// TwinCAT 3 PLC project PlanarTrackMovement_1
// ProgramVersion: 3.1.4026.12
// libraries:
//   HelperFunctions, * (Amazon)
//   RingBuffer, * (Amazon)
//   Tc2_Standard, * (Beckhoff Automation GmbH)
//   Tc2_System, * (Beckhoff Automation GmbH)
//   Tc2_Utilities, * (Beckhoff Automation GmbH)
//   Tc3_Mc3PlanarMotion, * (Beckhoff Automation GmbH)
//   Tc3_Module, * (Beckhoff Automation GmbH)
//   Tc3_Physics, * (Beckhoff Automation GmbH)
//   Tc3_XTS_Utility, * (Beckhoff Automation GmbH)
// project tree:
//   DUTs/ E_MergeType.TcDUT, E_TrackNum.TcDUT, MoverSort.TcDUT, ST_Debounce.TcDUT, ST_MoverOptions.TcDUT, ST_PlanarTrackConfig.TcDUT, ST_DivertConfig.TcDUT, ST_ExpMoverStatus.TcDUT, ST_PlcSystem.TcDUT, ST_SectorsConfig.TcDUT, ST_SectorsStatus.TcDUT, ST_SwitchStatus.TcDUT, ST_SectorConfig.TcDUT, ST_SectorStatus.TcDUT, ST_ShortcutConfig.TcDUT, ST_SwitchConfig.TcDUT, ST_TrackConfig.TcDUT, ST_MoverConfig.TcDUT
//   GVLs/ GC.TcGVL, GVL_General.TcGVL, GVL_Mc3.TcGVL
//   ITFs/ I_Mover.TcIO, I_MoverSector.TcIO
//   / PlcTask.TcTTO
//   POUs/FBs/ FB_AllTrackSectors.TcPOU, FB_AllExpMovers.TcPOU, FB_DivertQueue.TcPOU, FB_ExpandedMover.TcPOU, FB_MoverLists.TcPOU, FB_MoveState.TcPOU, FB_RobMover.TcPOU (excluded from build), FB_PlanarXtsMover.TcPOU, FB_PWM.TcPOU (not stored), FB_TrackSector.TcPOU, FB_SwitchMagnet.TcPOU, FB_TrackSectors.TcPOU, ReadTcCom.TcPOU
//   POUs/FUNs/ F_CurrentVelocity.TcPOU, F_PosnInitial.TcPOU, F_PosnDisp.TcPOU, F_t_SL2a.TcPOU, F_t_v0.TcPOU, F_t_vConstant.TcPOU, IsBetween.TcPOU (not stored), PositionF_CurrentCoeff.TcPOU
//   POUs/ MAIN.TcPOU
// real-time tasks:
//   TASK XTS Task: cycle T#500us, priority 1, ADS port 350
//   TASK Job Task: cycle default, priority 32
//   TASK MC-Task (MET): cycle T#2ms, priority 3, ADS port 521
//   TASK MC-Task (MPT): cycle T#10ms, priority 8, ADS port 531
//   TASK PlcTask: cycle T#1ms, priority 20, ADS port 351
//   TASK PlcTask1: cycle T#1ms, priority 21, ADS port 352
// motion (NC):
//   TASK NC-Task 1 SAF: cycle T#2ms, priority 4, ADS port 501
//   TASK NC-Task 1 SVB: cycle T#10ms, priority 9, ADS port 511
//   AXIS Axis 1 (id 1)
//     General: UnitFlags=#x00000004
//     Dynamic: Acceleration=4000, Deceleration=4000, Jerk=10000
//     Velo: FastManual=1200, Maximum=5000
//     OtherSettings: AllowMotionCmdToSlave=true
//     encoder EncType=28
//       EncPara: MaxCount=#xffffffff
//     drive DrvType=22
//       DrvPara: MaxCount=#xffffffff, DriveControlDWord=#x00000100
//         Analog: VeloReferenz=5000, TorqueSetpointScale=10, ScaleFactorActTorque=0.1
//         TimeComp: TaskDelayCycles=1
//     controller CtrType=1
//       CtrPara: PriorControlFactor=1
//         PosDiffControl: Range=50
//         Observer: BandWidth=20
// I/O:
//   DEVICE Device 1 (EtherCAT) (disabled), AmsNetId 11.200.5.30.2.1
//     Term 1 (EK1200) [EK1200-5000 EtherCAT Power supply (2A E-Bus)]
//       Term 2 (EL1809) [EL1809 16Ch. Dig. Input 24V, 3ms]
//       Term 3 (EL1018) [EL1018 8Ch. Dig. Input 24V, 10µs]
//       Term 4 (EL2809) [EL2809 16Ch. Dig. Output 24V, 0.5A]
//       Term 5 (EL3004) [EL3004 4Ch. Ana. Input +/-10V]
//       Term 6 (EL3314) [EL3314 4Ch. Ana. Input Thermocouple (TC)]
//       Term 7 (EL4034) [EL4034 4Ch. Ana. Output +/-10V, 12bit]
//       Term 8 (EL7062) [EL7062-0000 Stepper Drive]
//       Term 9 (EL9576) [EL9576 Brake chopper terminal]
//       Term 10 (EL9410) [EL9410 E-Bus Power Supplier  (Diagnostics)]
//       Term 11 (EL1904) [EL1904, 4 Ch. Safety Input 24V, TwinSAFE]
//         modules: Module 1 (FSOES)
//       Term 12 (EL1904) [EL1904, 4 Ch. Safety Input 24V, TwinSAFE]
//         modules: Module 1 (FSOES)
//       Term 13 (EL2912) [EL2912, 2Ch. Safety Output 24V, 2A, TwinSAFE]
//         modules: Module 2 (FSOUT), Module 3 (DEVICEIO), Module 4 (FSLOGIC)
//       Term 14 (EK1122) [EK1122 2 port EtherCAT junction]
//       Term 95 (EL6695) [EL6695 EtherCAT Bridge terminal (Primary)]
//       Term 16 (EK1110) [EK1110 EtherCAT extension]
//     Term 15 (AX8640-0000-0105) [AX8640-0000-0105]
//       startup 32768:16 := 12 // PSM Parameters / Ext brake resistor overload factor at 1% duty cycle
//       startup 32768:18 := 21DCC63E // PSM Parameters / External brake resistor time constant 1
//       startup 32768:19 := C37C6442 // PSM Parameters / External brake resistor time constant 2
//       startup 32768:20 := 8CA3E13F // PSM Parameters / External brake resistor partial fraction factor
//   DEVICE Device 8 (EtherCAT) (disabled), AmsNetId 11.200.5.30.9.1
//     Box 18 (AT5100-0100) [AT5100-0100 XTS XL, TwinSAFE]
//       modules: Module 1 (SAFETY)
//     Box 19 (AT5100-0100) [AT5100-0100 XTS XL, TwinSAFE]
//       modules: Module 1 (SAFETY)
//     Box 20 (AT5100-0100) [AT5100-0100 XTS XL, TwinSAFE]
//       modules: Module 1 (SAFETY)
//     Box 21 (AT5100-0100) [AT5100-0100 XTS XL, TwinSAFE]
//       modules: Module 1 (SAFETY)
//     Box 22 (AT5100-0100) [AT5100-0100 XTS XL, TwinSAFE]
//       modules: Module 1 (SAFETY)
//     Box 23 (AT5100-0100) [AT5100-0100 XTS XL, TwinSAFE]
//       modules: Module 1 (SAFETY)
//     Box 24 (AT5100-0100) [AT5100-0100 XTS XL, TwinSAFE]
//       modules: Module 1 (SAFETY)
//     Box 25 (AT5100-0100) [AT5100-0100 XTS XL, TwinSAFE]
//       modules: Module 1 (SAFETY)
//     Box 26 (AT5100-0100) [AT5100-0100 XTS XL, TwinSAFE]
//       modules: Module 1 (SAFETY)
//     Box 27 (AT5100-0100) [AT5100-0100 XTS XL, TwinSAFE]
//       modules: Module 1 (SAFETY)
//     Box 28 (AT5100-0100) [AT5100-0100 XTS XL, TwinSAFE]
//       modules: Module 1 (SAFETY)
//     Box 29 (AT5100-0100) [AT5100-0100 XTS XL, TwinSAFE]
//       modules: Module 1 (SAFETY)
//     Box 30 (AT5100-0100) [AT5100-0100 XTS XL, TwinSAFE]
//       modules: Module 1 (SAFETY)
//     Box 31 (AT5100-0100) [AT5100-0100 XTS XL, TwinSAFE]
//       modules: Module 1 (SAFETY)
//     Box 32 (AT5100-0100) [AT5100-0100 XTS XL, TwinSAFE]
//       modules: Module 1 (SAFETY)
//     Box 33 (AT5100-0100) [AT5100-0100 XTS XL, TwinSAFE]
//       modules: Module 1 (SAFETY)
//     Box 34 (AT5100-0100) [AT5100-0100 XTS XL, TwinSAFE]
//       modules: Module 1 (SAFETY)
//     Box 35 (AT5100-0100) [AT5100-0100 XTS XL, TwinSAFE]
//       modules: Module 1 (SAFETY)
//     Box 36 (AT5100-0100) [AT5100-0100 XTS XL, TwinSAFE]
//       modules: Module 1 (SAFETY)
//     Box 37 (AT5100-0100) [AT5100-0100 XTS XL, TwinSAFE]
//       modules: Module 1 (SAFETY)
//     Box 38 (AT5100-0100) [AT5100-0100 XTS XL, TwinSAFE]
//       modules: Module 1 (SAFETY)
//     Box 39 (AT5100-0100) [AT5100-0100 XTS XL, TwinSAFE]
//       modules: Module 1 (SAFETY)
//     Box 40 (AT5100-0100) [AT5100-0100 XTS XL, TwinSAFE]
//       modules: Module 1 (SAFETY)
//     Box 41 (AT5100-0100) [AT5100-0100 XTS XL, TwinSAFE]
//       modules: Module 1 (SAFETY)
//     Box 42 (AT5100-0100) [AT5100-0100 XTS XL, TwinSAFE]
//       modules: Module 1 (SAFETY)
//     Box 43 (AT5100-0100) [AT5100-0100 XTS XL, TwinSAFE]
//       modules: Module 1 (SAFETY)
//     Box 44 (AT5100-0100) [AT5100-0100 XTS XL, TwinSAFE]
//       modules: Module 1 (SAFETY)
//     Box 45 (AT5100-0100) [AT5100-0100 XTS XL, TwinSAFE]
//       modules: Module 1 (SAFETY)
//     Box 46 (AT5100-0100) [AT5100-0100 XTS XL, TwinSAFE]
//       modules: Module 1 (SAFETY)
//     Box 47 (AT5100-0100) [AT5100-0100 XTS XL, TwinSAFE]
//       modules: Module 1 (SAFETY)
//     Box 48 (AT5100-0100) [AT5100-0100 XTS XL, TwinSAFE]
//       modules: Module 1 (SAFETY)
//     Box 49 (AT5100-0100) [AT5100-0100 XTS XL, TwinSAFE]
//       modules: Module 1 (SAFETY)
//   DEVICE Device 4 (EtherCAT) (disabled), AmsNetId 11.200.5.30.5.1
//     Box 50 (AT5100-0100) [AT5100-0100 XTS XL, TwinSAFE]
//       modules: Module 1 (SAFETY)
//     Box 51 (AT5100-0100) [AT5100-0100 XTS XL, TwinSAFE]
//       modules: Module 1 (SAFETY)
//     Box 52 (AT5100-0100) [AT5100-0100 XTS XL, TwinSAFE]
//       modules: Module 1 (SAFETY)
//     Box 53 (AT5100-0100) [AT5100-0100 XTS XL, TwinSAFE]
//       modules: Module 1 (SAFETY)
//     Box 54 (AT5100-0100) [AT5100-0100 XTS XL, TwinSAFE]
//       modules: Module 1 (SAFETY)
//     Box 55 (AT5100-0100) [AT5100-0100 XTS XL, TwinSAFE]
//       modules: Module 1 (SAFETY)
//     Box 56 (AT5100-0100) [AT5100-0100 XTS XL, TwinSAFE]
//       modules: Module 1 (SAFETY)
//     Box 57 (AT5100-0100) [AT5100-0100 XTS XL, TwinSAFE]
//       modules: Module 1 (SAFETY)
//     Box 58 (AT5100-0100) [AT5100-0100 XTS XL, TwinSAFE]
//       modules: Module 1 (SAFETY)
//     Box 59 (AT5100-0100) [AT5100-0100 XTS XL, TwinSAFE]
//       modules: Module 1 (SAFETY)
//     Box 60 (AT5100-0100) [AT5100-0100 XTS XL, TwinSAFE]
//       modules: Module 1 (SAFETY)
//     Box 61 (AT5100-0100) [AT5100-0100 XTS XL, TwinSAFE]
//       modules: Module 1 (SAFETY)
//     Box 62 (AT5100-0100) [AT5100-0100 XTS XL, TwinSAFE]
//       modules: Module 1 (SAFETY)
//     Box 63 (AT5100-0100) [AT5100-0100 XTS XL, TwinSAFE]
//       modules: Module 1 (SAFETY)
//     Box 64 (AT5100-0100) [AT5100-0100 XTS XL, TwinSAFE]
//       modules: Module 1 (SAFETY)
//     Box 65 (AT5100-0100) [AT5100-0100 XTS XL, TwinSAFE]
//       modules: Module 1 (SAFETY)
//     Box 66 (AT5100-0100) [AT5100-0100 XTS XL, TwinSAFE]
//       modules: Module 1 (SAFETY)
//     Box 67 (AT5100-0100) [AT5100-0100 XTS XL, TwinSAFE]
//       modules: Module 1 (SAFETY)
//     Box 68 (AT5100-0100) [AT5100-0100 XTS XL, TwinSAFE]
//       modules: Module 1 (SAFETY)
//     Box 69 (AT5100-0100) [AT5100-0100 XTS XL, TwinSAFE]
//       modules: Module 1 (SAFETY)
//     Box 70 (AT5100-0100) [AT5100-0100 XTS XL, TwinSAFE]
//       modules: Module 1 (SAFETY)
//     Box 71 (AT5100-0100) [AT5100-0100 XTS XL, TwinSAFE]
//       modules: Module 1 (SAFETY)
//     Box 72 (AT5100-0100) [AT5100-0100 XTS XL, TwinSAFE]
//       modules: Module 1 (SAFETY)
//     Box 73 (AT5100-0100) [AT5100-0100 XTS XL, TwinSAFE]
//       modules: Module 1 (SAFETY)
//     Box 74 (AT5100-0100) [AT5100-0100 XTS XL, TwinSAFE]
//       modules: Module 1 (SAFETY)
//     Box 75 (AT5100-0100) [AT5100-0100 XTS XL, TwinSAFE]
//       modules: Module 1 (SAFETY)
//     Box 76 (AT5100-0100) [AT5100-0100 XTS XL, TwinSAFE]
//       modules: Module 1 (SAFETY)
//     Box 77 (AT5100-0100) [AT5100-0100 XTS XL, TwinSAFE]
//       modules: Module 1 (SAFETY)
//     Box 78 (AT5100-0100) [AT5100-0100 XTS XL, TwinSAFE]
//       modules: Module 1 (SAFETY)
//     Box 79 (AT5100-0100) [AT5100-0100 XTS XL, TwinSAFE]
//       modules: Module 1 (SAFETY)
//     Box 80 (AT5100-0100) [AT5100-0100 XTS XL, TwinSAFE]
//       modules: Module 1 (SAFETY)
//     Box 81 (AT5100-0100) [AT5100-0100 XTS XL, TwinSAFE]
//       modules: Module 1 (SAFETY)
// variable links:
//   Device 1 (EtherCAT) <-> Device 1 (EtherCAT)/Term 1 (EK1200)/Term 12 (EL1904)
//     Term 1 (EK1200)/Term 13 (EL2912)/ConnectionInputs/TwinSafeGroup1.Term 12 (EL1904) - Module 1 (FSOES)_144 TxPDO <-> Module 1 (FSOES)/RxPDO/FSOE
//   Device 1 (EtherCAT) <-> Device 1 (EtherCAT)/Term 1 (EK1200)/Term 13 (EL2912)
//     Term 1 (EK1200)/Term 11 (EL1904)/Module 1 (FSOES)/RxPDO/FSOE <-> ConnectionInputs/TwinSafeGroup1.Term 11 (EL1904) - Module 1 (FSOES)_4 TxPDO
//     Term 1 (EK1200)/Term 11 (EL1904)/Module 1 (FSOES)/TxPDO/FSOE <-> ConnectionOutputs/TwinSafeGroup1.Term 11 (EL1904) - Module 1 (FSOES)_4 RxPDO
//     Term 1 (EK1200)/Term 12 (EL1904)/Module 1 (FSOES)/TxPDO/FSOE <-> ConnectionOutputs/TwinSafeGroup1.Term 12 (EL1904) - Module 1 (FSOES)_144 RxPDO
//   Device 1 (EtherCAT) <-> Device 4 (EtherCAT)/Box 50 (AT5100-0100)
//     Term 1 (EK1200)/Term 13 (EL2912)/ConnectionInputs/TwinSafeGroup1.Box 50 (AT5100-0100) - Module 1 (SAFETY)_107 TxPDO <-> Module 1 (SAFETY)/SAFETY FSoE Connection 1 Receive Message/Message_4
//     Term 1 (EK1200)/Term 13 (EL2912)/ConnectionOutputs/TwinSafeGroup1.Box 50 (AT5100-0100) - Module 1 (SAFETY)_107 RxPDO <-> Module 1 (SAFETY)/SAFETY FSoE Connection 1 Send Message/Message_4
//   Device 1 (EtherCAT) <-> Device 4 (EtherCAT)/Box 51 (AT5100-0100)
//     Term 1 (EK1200)/Term 13 (EL2912)/ConnectionInputs/TwinSafeGroup1.Box 51 (AT5100-0100) - Module 1 (SAFETY)_108 TxPDO <-> Module 1 (SAFETY)/SAFETY FSoE Connection 1 Receive Message/Message_4
//     Term 1 (EK1200)/Term 13 (EL2912)/ConnectionOutputs/TwinSafeGroup1.Box 51 (AT5100-0100) - Module 1 (SAFETY)_108 RxPDO <-> Module 1 (SAFETY)/SAFETY FSoE Connection 1 Send Message/Message_4
//   Device 1 (EtherCAT) <-> Device 4 (EtherCAT)/Box 52 (AT5100-0100)
//     Term 1 (EK1200)/Term 13 (EL2912)/ConnectionInputs/TwinSafeGroup1.Box 52 (AT5100-0100) - Module 1 (SAFETY)_109 TxPDO <-> Module 1 (SAFETY)/SAFETY FSoE Connection 1 Receive Message/Message_4
//     Term 1 (EK1200)/Term 13 (EL2912)/ConnectionOutputs/TwinSafeGroup1.Box 52 (AT5100-0100) - Module 1 (SAFETY)_109 RxPDO <-> Module 1 (SAFETY)/SAFETY FSoE Connection 1 Send Message/Message_4
//   Device 1 (EtherCAT) <-> Device 4 (EtherCAT)/Box 53 (AT5100-0100)
//     Term 1 (EK1200)/Term 13 (EL2912)/ConnectionInputs/TwinSafeGroup1.Box 53 (AT5100-0100) - Module 1 (SAFETY)_110 TxPDO <-> Module 1 (SAFETY)/SAFETY FSoE Connection 1 Receive Message/Message_4
//     Term 1 (EK1200)/Term 13 (EL2912)/ConnectionOutputs/TwinSafeGroup1.Box 53 (AT5100-0100) - Module 1 (SAFETY)_110 RxPDO <-> Module 1 (SAFETY)/SAFETY FSoE Connection 1 Send Message/Message_4
//   Device 1 (EtherCAT) <-> Device 4 (EtherCAT)/Box 54 (AT5100-0100)
//     Term 1 (EK1200)/Term 13 (EL2912)/ConnectionInputs/TwinSafeGroup1.Box 54 (AT5100-0100) - Module 1 (SAFETY)_111 TxPDO <-> Module 1 (SAFETY)/SAFETY FSoE Connection 1 Receive Message/Message_4
//     Term 1 (EK1200)/Term 13 (EL2912)/ConnectionOutputs/TwinSafeGroup1.Box 54 (AT5100-0100) - Module 1 (SAFETY)_111 RxPDO <-> Module 1 (SAFETY)/SAFETY FSoE Connection 1 Send Message/Message_4
//   Device 1 (EtherCAT) <-> Device 4 (EtherCAT)/Box 55 (AT5100-0100)
//     Term 1 (EK1200)/Term 13 (EL2912)/ConnectionInputs/TwinSafeGroup1.Box 55 (AT5100-0100) - Module 1 (SAFETY)_112 TxPDO <-> Module 1 (SAFETY)/SAFETY FSoE Connection 1 Receive Message/Message_4
//     Term 1 (EK1200)/Term 13 (EL2912)/ConnectionOutputs/TwinSafeGroup1.Box 55 (AT5100-0100) - Module 1 (SAFETY)_112 RxPDO <-> Module 1 (SAFETY)/SAFETY FSoE Connection 1 Send Message/Message_4
//   Device 1 (EtherCAT) <-> Device 4 (EtherCAT)/Box 56 (AT5100-0100)
//     Term 1 (EK1200)/Term 13 (EL2912)/ConnectionInputs/TwinSafeGroup1.Box 56 (AT5100-0100) - Module 1 (SAFETY)_113 TxPDO <-> Module 1 (SAFETY)/SAFETY FSoE Connection 1 Receive Message/Message_4
//     Term 1 (EK1200)/Term 13 (EL2912)/ConnectionOutputs/TwinSafeGroup1.Box 56 (AT5100-0100) - Module 1 (SAFETY)_113 RxPDO <-> Module 1 (SAFETY)/SAFETY FSoE Connection 1 Send Message/Message_4
//   Device 1 (EtherCAT) <-> Device 4 (EtherCAT)/Box 57 (AT5100-0100)
//     Term 1 (EK1200)/Term 13 (EL2912)/ConnectionInputs/TwinSafeGroup1.Box 57 (AT5100-0100) - Module 1 (SAFETY)_114 TxPDO <-> Module 1 (SAFETY)/SAFETY FSoE Connection 1 Receive Message/Message_4
//     Term 1 (EK1200)/Term 13 (EL2912)/ConnectionOutputs/TwinSafeGroup1.Box 57 (AT5100-0100) - Module 1 (SAFETY)_114 RxPDO <-> Module 1 (SAFETY)/SAFETY FSoE Connection 1 Send Message/Message_4
//   Device 1 (EtherCAT) <-> Device 4 (EtherCAT)/Box 58 (AT5100-0100)
//     Term 1 (EK1200)/Term 13 (EL2912)/ConnectionInputs/TwinSafeGroup1.Box 58 (AT5100-0100) - Module 1 (SAFETY)_115 TxPDO <-> Module 1 (SAFETY)/SAFETY FSoE Connection 1 Receive Message/Message_4
//     Term 1 (EK1200)/Term 13 (EL2912)/ConnectionOutputs/TwinSafeGroup1.Box 58 (AT5100-0100) - Module 1 (SAFETY)_115 RxPDO <-> Module 1 (SAFETY)/SAFETY FSoE Connection 1 Send Message/Message_4
//   Device 1 (EtherCAT) <-> Device 4 (EtherCAT)/Box 59 (AT5100-0100)
//     Term 1 (EK1200)/Term 13 (EL2912)/ConnectionOutputs/TwinSafeGroup1.Box 59 (AT5100-0100) - Module 1 (SAFETY)_116 RxPDO <-> Module 1 (SAFETY)/SAFETY FSoE Connection 1 Send Message/Message_4
//   Device 1 (EtherCAT) <-> Device 4 (EtherCAT)/Box 60 (AT5100-0100)
//     Term 1 (EK1200)/Term 13 (EL2912)/ConnectionInputs/TwinSafeGroup1.Box 60 (AT5100-0100) - Module 1 (SAFETY)_117 TxPDO <-> Module 1 (SAFETY)/SAFETY FSoE Connection 1 Receive Message/Message_4
//     Term 1 (EK1200)/Term 13 (EL2912)/ConnectionOutputs/TwinSafeGroup1.Box 60 (AT5100-0100) - Module 1 (SAFETY)_117 RxPDO <-> Module 1 (SAFETY)/SAFETY FSoE Connection 1 Send Message/Message_4
//   Device 1 (EtherCAT) <-> Device 4 (EtherCAT)/Box 61 (AT5100-0100)
//     Term 1 (EK1200)/Term 13 (EL2912)/ConnectionInputs/TwinSafeGroup1.Box 61 (AT5100-0100) - Module 1 (SAFETY)_118 TxPDO <-> Module 1 (SAFETY)/SAFETY FSoE Connection 1 Receive Message/Message_4
//   Device 1 (EtherCAT) <-> Device 4 (EtherCAT)/Box 62 (AT5100-0100)
//     Term 1 (EK1200)/Term 13 (EL2912)/ConnectionInputs/TwinSafeGroup1.Box 62 (AT5100-0100) - Module 1 (SAFETY)_119 TxPDO <-> Module 1 (SAFETY)/SAFETY FSoE Connection 1 Receive Message/Message_4
//   Device 1 (EtherCAT) <-> Device 4 (EtherCAT)/Box 63 (AT5100-0100)
//     Term 1 (EK1200)/Term 13 (EL2912)/ConnectionInputs/TwinSafeGroup1.Box 63 (AT5100-0100) - Module 1 (SAFETY)_120 TxPDO <-> Module 1 (SAFETY)/SAFETY FSoE Connection 1 Receive Message/Message_4
//     Term 1 (EK1200)/Term 13 (EL2912)/ConnectionOutputs/TwinSafeGroup1.Box 63 (AT5100-0100) - Module 1 (SAFETY)_120 RxPDO <-> Module 1 (SAFETY)/SAFETY FSoE Connection 1 Send Message/Message_4
//   Device 1 (EtherCAT) <-> Device 4 (EtherCAT)/Box 64 (AT5100-0100)
//     Term 1 (EK1200)/Term 13 (EL2912)/ConnectionInputs/TwinSafeGroup1.Box 64 (AT5100-0100) - Module 1 (SAFETY)_121 TxPDO <-> Module 1 (SAFETY)/SAFETY FSoE Connection 1 Receive Message/Message_4
//     Term 1 (EK1200)/Term 13 (EL2912)/ConnectionOutputs/TwinSafeGroup1.Box 64 (AT5100-0100) - Module 1 (SAFETY)_121 RxPDO <-> Module 1 (SAFETY)/SAFETY FSoE Connection 1 Send Message/Message_4
//   Device 1 (EtherCAT) <-> Device 4 (EtherCAT)/Box 65 (AT5100-0100)
//     Term 1 (EK1200)/Term 13 (EL2912)/ConnectionInputs/TwinSafeGroup1.Box 65 (AT5100-0100) - Module 1 (SAFETY)_122 TxPDO <-> Module 1 (SAFETY)/SAFETY FSoE Connection 1 Receive Message/Message_4
//     Term 1 (EK1200)/Term 13 (EL2912)/ConnectionOutputs/TwinSafeGroup1.Box 65 (AT5100-0100) - Module 1 (SAFETY)_122 RxPDO <-> Module 1 (SAFETY)/SAFETY FSoE Connection 1 Send Message/Message_4
//   Device 1 (EtherCAT) <-> Device 4 (EtherCAT)/Box 66 (AT5100-0100)
//     Term 1 (EK1200)/Term 13 (EL2912)/ConnectionInputs/TwinSafeGroup1.Box 66 (AT5100-0100) - Module 1 (SAFETY)_123 TxPDO <-> Module 1 (SAFETY)/SAFETY FSoE Connection 1 Receive Message/Message_4
//     Term 1 (EK1200)/Term 13 (EL2912)/ConnectionOutputs/TwinSafeGroup1.Box 66 (AT5100-0100) - Module 1 (SAFETY)_123 RxPDO <-> Module 1 (SAFETY)/SAFETY FSoE Connection 1 Send Message/Message_4
//   Device 1 (EtherCAT) <-> Device 4 (EtherCAT)/Box 67 (AT5100-0100)
//     Term 1 (EK1200)/Term 13 (EL2912)/ConnectionInputs/TwinSafeGroup1.Box 67 (AT5100-0100) - Module 1 (SAFETY)_124 TxPDO <-> Module 1 (SAFETY)/SAFETY FSoE Connection 1 Receive Message/Message_4
//     Term 1 (EK1200)/Term 13 (EL2912)/ConnectionOutputs/TwinSafeGroup1.Box 67 (AT5100-0100) - Module 1 (SAFETY)_124 RxPDO <-> Module 1 (SAFETY)/SAFETY FSoE Connection 1 Send Message/Message_4
//   Device 1 (EtherCAT) <-> Device 4 (EtherCAT)/Box 68 (AT5100-0100)
//     Term 1 (EK1200)/Term 13 (EL2912)/ConnectionInputs/TwinSafeGroup1.Box 68 (AT5100-0100) - Module 1 (SAFETY)_125 TxPDO <-> Module 1 (SAFETY)/SAFETY FSoE Connection 1 Receive Message/Message_4
//     Term 1 (EK1200)/Term 13 (EL2912)/ConnectionOutputs/TwinSafeGroup1.Box 68 (AT5100-0100) - Module 1 (SAFETY)_125 RxPDO <-> Module 1 (SAFETY)/SAFETY FSoE Connection 1 Send Message/Message_4
//   Device 1 (EtherCAT) <-> Device 4 (EtherCAT)/Box 69 (AT5100-0100)
//     Term 1 (EK1200)/Term 13 (EL2912)/ConnectionInputs/TwinSafeGroup1.Box 69 (AT5100-0100) - Module 1 (SAFETY)_126 TxPDO <-> Module 1 (SAFETY)/SAFETY FSoE Connection 1 Receive Message/Message_4
//     Term 1 (EK1200)/Term 13 (EL2912)/ConnectionOutputs/TwinSafeGroup1.Box 69 (AT5100-0100) - Module 1 (SAFETY)_126 RxPDO <-> Module 1 (SAFETY)/SAFETY FSoE Connection 1 Send Message/Message_4
//   Device 1 (EtherCAT) <-> Device 4 (EtherCAT)/Box 70 (AT5100-0100)
//     Term 1 (EK1200)/Term 13 (EL2912)/ConnectionInputs/TwinSafeGroup1.Box 70 (AT5100-0100) - Module 1 (SAFETY)_127 TxPDO <-> Module 1 (SAFETY)/SAFETY FSoE Connection 1 Receive Message/Message_4
//     Term 1 (EK1200)/Term 13 (EL2912)/ConnectionOutputs/TwinSafeGroup1.Box 70 (AT5100-0100) - Module 1 (SAFETY)_127 RxPDO <-> Module 1 (SAFETY)/SAFETY FSoE Connection 1 Send Message/Message_4
//   Device 1 (EtherCAT) <-> Device 4 (EtherCAT)/Box 71 (AT5100-0100)
//     Term 1 (EK1200)/Term 13 (EL2912)/ConnectionInputs/TwinSafeGroup1.Box 71 (AT5100-0100) - Module 1 (SAFETY)_128 TxPDO <-> Module 1 (SAFETY)/SAFETY FSoE Connection 1 Receive Message/Message_4
//     Term 1 (EK1200)/Term 13 (EL2912)/ConnectionOutputs/TwinSafeGroup1.Box 71 (AT5100-0100) - Module 1 (SAFETY)_128 RxPDO <-> Module 1 (SAFETY)/SAFETY FSoE Connection 1 Send Message/Message_4
//   Device 1 (EtherCAT) <-> Device 4 (EtherCAT)/Box 72 (AT5100-0100)
//     Term 1 (EK1200)/Term 13 (EL2912)/ConnectionInputs/TwinSafeGroup1.Box 72 (AT5100-0100) - Module 1 (SAFETY)_129 TxPDO <-> Module 1 (SAFETY)/SAFETY FSoE Connection 1 Receive Message/Message_4
//     Term 1 (EK1200)/Term 13 (EL2912)/ConnectionOutputs/TwinSafeGroup1.Box 72 (AT5100-0100) - Module 1 (SAFETY)_129 RxPDO <-> Module 1 (SAFETY)/SAFETY FSoE Connection 1 Send Message/Message_4
//   Device 1 (EtherCAT) <-> Device 4 (EtherCAT)/Box 73 (AT5100-0100)
//     Term 1 (EK1200)/Term 13 (EL2912)/ConnectionInputs/TwinSafeGroup1.Box 73 (AT5100-0100) - Module 1 (SAFETY)_130 TxPDO <-> Module 1 (SAFETY)/SAFETY FSoE Connection 1 Receive Message/Message_4
//     Term 1 (EK1200)/Term 13 (EL2912)/ConnectionOutputs/TwinSafeGroup1.Box 73 (AT5100-0100) - Module 1 (SAFETY)_130 RxPDO <-> Module 1 (SAFETY)/SAFETY FSoE Connection 1 Send Message/Message_4
//   Device 1 (EtherCAT) <-> Device 4 (EtherCAT)/Box 74 (AT5100-0100)
//     Term 1 (EK1200)/Term 13 (EL2912)/ConnectionOutputs/TwinSafeGroup1.Box 74 (AT5100-0100) - Module 1 (SAFETY)_131 RxPDO <-> Module 1 (SAFETY)/SAFETY FSoE Connection 1 Send Message/Message_4
//   Device 1 (EtherCAT) <-> Device 4 (EtherCAT)/Box 75 (AT5100-0100)
//     Term 1 (EK1200)/Term 13 (EL2912)/ConnectionInputs/TwinSafeGroup1.Box 75 (AT5100-0100) - Module 1 (SAFETY)_132 TxPDO <-> Module 1 (SAFETY)/SAFETY FSoE Connection 1 Receive Message/Message_4
//     Term 1 (EK1200)/Term 13 (EL2912)/ConnectionOutputs/TwinSafeGroup1.Box 75 (AT5100-0100) - Module 1 (SAFETY)_132 RxPDO <-> Module 1 (SAFETY)/SAFETY FSoE Connection 1 Send Message/Message_4
//   Device 1 (EtherCAT) <-> Device 4 (EtherCAT)/Box 76 (AT5100-0100)
//     Term 1 (EK1200)/Term 13 (EL2912)/ConnectionInputs/TwinSafeGroup1.Box 76 (AT5100-0100) - Module 1 (SAFETY)_133 TxPDO <-> Module 1 (SAFETY)/SAFETY FSoE Connection 1 Receive Message/Message_4
//     Term 1 (EK1200)/Term 13 (EL2912)/ConnectionOutputs/TwinSafeGroup1.Box 76 (AT5100-0100) - Module 1 (SAFETY)_133 RxPDO <-> Module 1 (SAFETY)/SAFETY FSoE Connection 1 Send Message/Message_4
//   Device 1 (EtherCAT) <-> Device 4 (EtherCAT)/Box 77 (AT5100-0100)
//     Term 1 (EK1200)/Term 13 (EL2912)/ConnectionInputs/TwinSafeGroup1.Box 77 (AT5100-0100) - Module 1 (SAFETY)_134 TxPDO <-> Module 1 (SAFETY)/SAFETY FSoE Connection 1 Receive Message/Message_4
//     Term 1 (EK1200)/Term 13 (EL2912)/ConnectionOutputs/TwinSafeGroup1.Box 77 (AT5100-0100) - Module 1 (SAFETY)_134 RxPDO <-> Module 1 (SAFETY)/SAFETY FSoE Connection 1 Send Message/Message_4
//   Device 1 (EtherCAT) <-> Device 4 (EtherCAT)/Box 78 (AT5100-0100)
//     Term 1 (EK1200)/Term 13 (EL2912)/ConnectionInputs/TwinSafeGroup1.Box 78 (AT5100-0100) - Module 1 (SAFETY)_135 TxPDO <-> Module 1 (SAFETY)/SAFETY FSoE Connection 1 Receive Message/Message_4
//     Term 1 (EK1200)/Term 13 (EL2912)/ConnectionOutputs/TwinSafeGroup1.Box 78 (AT5100-0100) - Module 1 (SAFETY)_135 RxPDO <-> Module 1 (SAFETY)/SAFETY FSoE Connection 1 Send Message/Message_4
//   Device 1 (EtherCAT) <-> Device 4 (EtherCAT)/Box 79 (AT5100-0100)
//     Term 1 (EK1200)/Term 13 (EL2912)/ConnectionInputs/TwinSafeGroup1.Box 79 (AT5100-0100) - Module 1 (SAFETY)_136 TxPDO <-> Module 1 (SAFETY)/SAFETY FSoE Connection 1 Receive Message/Message_4
//     Term 1 (EK1200)/Term 13 (EL2912)/ConnectionOutputs/TwinSafeGroup1.Box 79 (AT5100-0100) - Module 1 (SAFETY)_136 RxPDO <-> Module 1 (SAFETY)/SAFETY FSoE Connection 1 Send Message/Message_4
//   Device 1 (EtherCAT) <-> Device 4 (EtherCAT)/Box 80 (AT5100-0100)
//     Term 1 (EK1200)/Term 13 (EL2912)/ConnectionInputs/TwinSafeGroup1.Box 80 (AT5100-0100) - Module 1 (SAFETY)_137 TxPDO <-> Module 1 (SAFETY)/SAFETY FSoE Connection 1 Receive Message/Message_4
//     Term 1 (EK1200)/Term 13 (EL2912)/ConnectionOutputs/TwinSafeGroup1.Box 80 (AT5100-0100) - Module 1 (SAFETY)_137 RxPDO <-> Module 1 (SAFETY)/SAFETY FSoE Connection 1 Send Message/Message_4
//   Device 1 (EtherCAT) <-> Device 4 (EtherCAT)/Box 81 (AT5100-0100)
//     Term 1 (EK1200)/Term 13 (EL2912)/ConnectionInputs/TwinSafeGroup1.Box 81 (AT5100-0100) - Module 1 (SAFETY)_138 TxPDO <-> Module 1 (SAFETY)/SAFETY FSoE Connection 1 Receive Message/Message_4
//     Term 1 (EK1200)/Term 13 (EL2912)/ConnectionOutputs/TwinSafeGroup1.Box 81 (AT5100-0100) - Module 1 (SAFETY)_138 RxPDO <-> Module 1 (SAFETY)/SAFETY FSoE Connection 1 Send Message/Message_4
//   Device 1 (EtherCAT) <-> Device 8 (EtherCAT)/Box 18 (AT5100-0100)
//     Term 1 (EK1200)/Term 13 (EL2912)/ConnectionInputs/TwinSafeGroup1.Box 18 (AT5100-0100) - Module 1 (SAFETY)_71 TxPDO <-> Module 1 (SAFETY)/SAFETY FSoE Connection 1 Receive Message/Message_4
//     Term 1 (EK1200)/Term 13 (EL2912)/ConnectionOutputs/TwinSafeGroup1.Box 18 (AT5100-0100) - Module 1 (SAFETY)_71 RxPDO <-> Module 1 (SAFETY)/SAFETY FSoE Connection 1 Send Message/Message_4
//   Device 1 (EtherCAT) <-> Device 8 (EtherCAT)/Box 19 (AT5100-0100)
//     Term 1 (EK1200)/Term 13 (EL2912)/ConnectionInputs/TwinSafeGroup1.Box 19 (AT5100-0100) - Module 1 (SAFETY)_76 TxPDO <-> Module 1 (SAFETY)/SAFETY FSoE Connection 1 Receive Message/Message_4
//     Term 1 (EK1200)/Term 13 (EL2912)/ConnectionOutputs/TwinSafeGroup1.Box 19 (AT5100-0100) - Module 1 (SAFETY)_76 RxPDO <-> Module 1 (SAFETY)/SAFETY FSoE Connection 1 Send Message/Message_4
//   Device 1 (EtherCAT) <-> Device 8 (EtherCAT)/Box 20 (AT5100-0100)
//     Term 1 (EK1200)/Term 13 (EL2912)/ConnectionInputs/TwinSafeGroup1.Box 20 (AT5100-0100) - Module 1 (SAFETY)_77 TxPDO <-> Module 1 (SAFETY)/SAFETY FSoE Connection 1 Receive Message/Message_4
//     Term 1 (EK1200)/Term 13 (EL2912)/ConnectionOutputs/TwinSafeGroup1.Box 20 (AT5100-0100) - Module 1 (SAFETY)_77 RxPDO <-> Module 1 (SAFETY)/SAFETY FSoE Connection 1 Send Message/Message_4
//   Device 1 (EtherCAT) <-> Device 8 (EtherCAT)/Box 21 (AT5100-0100)
//     Term 1 (EK1200)/Term 13 (EL2912)/ConnectionInputs/TwinSafeGroup1.Box 21 (AT5100-0100) - Module 1 (SAFETY)_78 TxPDO <-> Module 1 (SAFETY)/SAFETY FSoE Connection 1 Receive Message/Message_4
//     Term 1 (EK1200)/Term 13 (EL2912)/ConnectionOutputs/TwinSafeGroup1.Box 21 (AT5100-0100) - Module 1 (SAFETY)_78 RxPDO <-> Module 1 (SAFETY)/SAFETY FSoE Connection 1 Send Message/Message_4
//   Device 1 (EtherCAT) <-> Device 8 (EtherCAT)/Box 22 (AT5100-0100)
//     Term 1 (EK1200)/Term 13 (EL2912)/ConnectionInputs/TwinSafeGroup1.Box 22 (AT5100-0100) - Module 1 (SAFETY)_79 TxPDO <-> Module 1 (SAFETY)/SAFETY FSoE Connection 1 Receive Message/Message_4
//     Term 1 (EK1200)/Term 13 (EL2912)/ConnectionOutputs/TwinSafeGroup1.Box 22 (AT5100-0100) - Module 1 (SAFETY)_79 RxPDO <-> Module 1 (SAFETY)/SAFETY FSoE Connection 1 Send Message/Message_4
//   Device 1 (EtherCAT) <-> Device 8 (EtherCAT)/Box 23 (AT5100-0100)
//     Term 1 (EK1200)/Term 13 (EL2912)/ConnectionInputs/TwinSafeGroup1.Box 23 (AT5100-0100) - Module 1 (SAFETY)_80 TxPDO <-> Module 1 (SAFETY)/SAFETY FSoE Connection 1 Receive Message/Message_4
//     Term 1 (EK1200)/Term 13 (EL2912)/ConnectionOutputs/TwinSafeGroup1.Box 23 (AT5100-0100) - Module 1 (SAFETY)_80 RxPDO <-> Module 1 (SAFETY)/SAFETY FSoE Connection 1 Send Message/Message_4
//   Device 1 (EtherCAT) <-> Device 8 (EtherCAT)/Box 24 (AT5100-0100)
//     Term 1 (EK1200)/Term 13 (EL2912)/ConnectionOutputs/TwinSafeGroup1.Box 24 (AT5100-0100) - Module 1 (SAFETY)_81 RxPDO <-> Module 1 (SAFETY)/SAFETY FSoE Connection 1 Send Message/Message_4
//   Device 1 (EtherCAT) <-> Device 8 (EtherCAT)/Box 25 (AT5100-0100)
//     Term 1 (EK1200)/Term 13 (EL2912)/ConnectionInputs/TwinSafeGroup1.Box 25 (AT5100-0100) - Module 1 (SAFETY)_82 TxPDO <-> Module 1 (SAFETY)/SAFETY FSoE Connection 1 Receive Message/Message_4
//     Term 1 (EK1200)/Term 13 (EL2912)/ConnectionOutputs/TwinSafeGroup1.Box 25 (AT5100-0100) - Module 1 (SAFETY)_82 RxPDO <-> Module 1 (SAFETY)/SAFETY FSoE Connection 1 Send Message/Message_4
//   Device 1 (EtherCAT) <-> Device 8 (EtherCAT)/Box 26 (AT5100-0100)
//     Term 1 (EK1200)/Term 13 (EL2912)/ConnectionInputs/TwinSafeGroup1.Box 26 (AT5100-0100) - Module 1 (SAFETY)_83 TxPDO <-> Module 1 (SAFETY)/SAFETY FSoE Connection 1 Receive Message/Message_4
//     Term 1 (EK1200)/Term 13 (EL2912)/ConnectionOutputs/TwinSafeGroup1.Box 26 (AT5100-0100) - Module 1 (SAFETY)_83 RxPDO <-> Module 1 (SAFETY)/SAFETY FSoE Connection 1 Send Message/Message_4
//   Device 1 (EtherCAT) <-> Device 8 (EtherCAT)/Box 27 (AT5100-0100)
//     Term 1 (EK1200)/Term 13 (EL2912)/ConnectionInputs/TwinSafeGroup1.Box 27 (AT5100-0100) - Module 1 (SAFETY)_84 TxPDO <-> Module 1 (SAFETY)/SAFETY FSoE Connection 1 Receive Message/Message_4
//     Term 1 (EK1200)/Term 13 (EL2912)/ConnectionOutputs/TwinSafeGroup1.Box 27 (AT5100-0100) - Module 1 (SAFETY)_84 RxPDO <-> Module 1 (SAFETY)/SAFETY FSoE Connection 1 Send Message/Message_4
//   Device 1 (EtherCAT) <-> Device 8 (EtherCAT)/Box 28 (AT5100-0100)
//     Term 1 (EK1200)/Term 13 (EL2912)/ConnectionInputs/TwinSafeGroup1.Box 28 (AT5100-0100) - Module 1 (SAFETY)_85 TxPDO <-> Module 1 (SAFETY)/SAFETY FSoE Connection 1 Receive Message/Message_4
//     Term 1 (EK1200)/Term 13 (EL2912)/ConnectionOutputs/TwinSafeGroup1.Box 28 (AT5100-0100) - Module 1 (SAFETY)_85 RxPDO <-> Module 1 (SAFETY)/SAFETY FSoE Connection 1 Send Message/Message_4
//   Device 1 (EtherCAT) <-> Device 8 (EtherCAT)/Box 29 (AT5100-0100)
//     Term 1 (EK1200)/Term 13 (EL2912)/ConnectionInputs/TwinSafeGroup1.Box 29 (AT5100-0100) - Module 1 (SAFETY)_86 TxPDO <-> Module 1 (SAFETY)/SAFETY FSoE Connection 1 Receive Message/Message_4
//     Term 1 (EK1200)/Term 13 (EL2912)/ConnectionOutputs/TwinSafeGroup1.Box 29 (AT5100-0100) - Module 1 (SAFETY)_86 RxPDO <-> Module 1 (SAFETY)/SAFETY FSoE Connection 1 Send Message/Message_4
//   Device 1 (EtherCAT) <-> Device 8 (EtherCAT)/Box 30 (AT5100-0100)
//     Term 1 (EK1200)/Term 13 (EL2912)/ConnectionInputs/TwinSafeGroup1.Box 30 (AT5100-0100) - Module 1 (SAFETY)_87 TxPDO <-> Module 1 (SAFETY)/SAFETY FSoE Connection 1 Receive Message/Message_4
//     Term 1 (EK1200)/Term 13 (EL2912)/ConnectionOutputs/TwinSafeGroup1.Box 30 (AT5100-0100) - Module 1 (SAFETY)_87 RxPDO <-> Module 1 (SAFETY)/SAFETY FSoE Connection 1 Send Message/Message_4
//   Device 1 (EtherCAT) <-> Device 8 (EtherCAT)/Box 31 (AT5100-0100)
//     Term 1 (EK1200)/Term 13 (EL2912)/ConnectionInputs/TwinSafeGroup1.Box 31 (AT5100-0100) - Module 1 (SAFETY)_88 TxPDO <-> Module 1 (SAFETY)/SAFETY FSoE Connection 1 Receive Message/Message_4
//     Term 1 (EK1200)/Term 13 (EL2912)/ConnectionOutputs/TwinSafeGroup1.Box 31 (AT5100-0100) - Module 1 (SAFETY)_88 RxPDO <-> Module 1 (SAFETY)/SAFETY FSoE Connection 1 Send Message/Message_4
//   Device 1 (EtherCAT) <-> Device 8 (EtherCAT)/Box 32 (AT5100-0100)
//     Term 1 (EK1200)/Term 13 (EL2912)/ConnectionInputs/TwinSafeGroup1.Box 32 (AT5100-0100) - Module 1 (SAFETY)_89 TxPDO <-> Module 1 (SAFETY)/SAFETY FSoE Connection 1 Receive Message/Message_4
//     Term 1 (EK1200)/Term 13 (EL2912)/ConnectionOutputs/TwinSafeGroup1.Box 32 (AT5100-0100) - Module 1 (SAFETY)_89 RxPDO <-> Module 1 (SAFETY)/SAFETY FSoE Connection 1 Send Message/Message_4
//   Device 1 (EtherCAT) <-> Device 8 (EtherCAT)/Box 33 (AT5100-0100)
//     Term 1 (EK1200)/Term 13 (EL2912)/ConnectionInputs/TwinSafeGroup1.Box 33 (AT5100-0100) - Module 1 (SAFETY)_90 TxPDO <-> Module 1 (SAFETY)/SAFETY FSoE Connection 1 Receive Message/Message_4
//     Term 1 (EK1200)/Term 13 (EL2912)/ConnectionOutputs/TwinSafeGroup1.Box 33 (AT5100-0100) - Module 1 (SAFETY)_90 RxPDO <-> Module 1 (SAFETY)/SAFETY FSoE Connection 1 Send Message/Message_4
//   Device 1 (EtherCAT) <-> Device 8 (EtherCAT)/Box 34 (AT5100-0100)
//     Term 1 (EK1200)/Term 13 (EL2912)/ConnectionInputs/TwinSafeGroup1.Box 34 (AT5100-0100) - Module 1 (SAFETY)_91 TxPDO <-> Module 1 (SAFETY)/SAFETY FSoE Connection 1 Receive Message/Message_4
//     Term 1 (EK1200)/Term 13 (EL2912)/ConnectionOutputs/TwinSafeGroup1.Box 34 (AT5100-0100) - Module 1 (SAFETY)_91 RxPDO <-> Module 1 (SAFETY)/SAFETY FSoE Connection 1 Send Message/Message_4
//   Device 1 (EtherCAT) <-> Device 8 (EtherCAT)/Box 35 (AT5100-0100)
//     Term 1 (EK1200)/Term 13 (EL2912)/ConnectionInputs/TwinSafeGroup1.Box 35 (AT5100-0100) - Module 1 (SAFETY)_92 TxPDO <-> Module 1 (SAFETY)/SAFETY FSoE Connection 1 Receive Message/Message_4
//     Term 1 (EK1200)/Term 13 (EL2912)/ConnectionOutputs/TwinSafeGroup1.Box 35 (AT5100-0100) - Module 1 (SAFETY)_92 RxPDO <-> Module 1 (SAFETY)/SAFETY FSoE Connection 1 Send Message/Message_4
//   Device 1 (EtherCAT) <-> Device 8 (EtherCAT)/Box 36 (AT5100-0100)
//     Term 1 (EK1200)/Term 13 (EL2912)/ConnectionInputs/TwinSafeGroup1.Box 36 (AT5100-0100) - Module 1 (SAFETY)_93 TxPDO <-> Module 1 (SAFETY)/SAFETY FSoE Connection 1 Receive Message/Message_4
//     Term 1 (EK1200)/Term 13 (EL2912)/ConnectionOutputs/TwinSafeGroup1.Box 36 (AT5100-0100) - Module 1 (SAFETY)_93 RxPDO <-> Module 1 (SAFETY)/SAFETY FSoE Connection 1 Send Message/Message_4
//   Device 1 (EtherCAT) <-> Device 8 (EtherCAT)/Box 37 (AT5100-0100)
//     Term 1 (EK1200)/Term 13 (EL2912)/ConnectionInputs/TwinSafeGroup1.Box 37 (AT5100-0100) - Module 1 (SAFETY)_94 TxPDO <-> Module 1 (SAFETY)/SAFETY FSoE Connection 1 Receive Message/Message_4
//     Term 1 (EK1200)/Term 13 (EL2912)/ConnectionOutputs/TwinSafeGroup1.Box 37 (AT5100-0100) - Module 1 (SAFETY)_94 RxPDO <-> Module 1 (SAFETY)/SAFETY FSoE Connection 1 Send Message/Message_4
//   Device 1 (EtherCAT) <-> Device 8 (EtherCAT)/Box 38 (AT5100-0100)
//     Term 1 (EK1200)/Term 13 (EL2912)/ConnectionInputs/TwinSafeGroup1.Box 38 (AT5100-0100) - Module 1 (SAFETY)_95 TxPDO <-> Module 1 (SAFETY)/SAFETY FSoE Connection 1 Receive Message/Message_4
//     Term 1 (EK1200)/Term 13 (EL2912)/ConnectionOutputs/TwinSafeGroup1.Box 38 (AT5100-0100) - Module 1 (SAFETY)_95 RxPDO <-> Module 1 (SAFETY)/SAFETY FSoE Connection 1 Send Message/Message_4
//   Device 1 (EtherCAT) <-> Device 8 (EtherCAT)/Box 39 (AT5100-0100)
//     Term 1 (EK1200)/Term 13 (EL2912)/ConnectionInputs/TwinSafeGroup1.Box 39 (AT5100-0100) - Module 1 (SAFETY)_96 TxPDO <-> Module 1 (SAFETY)/SAFETY FSoE Connection 1 Receive Message/Message_4
//     Term 1 (EK1200)/Term 13 (EL2912)/ConnectionOutputs/TwinSafeGroup1.Box 39 (AT5100-0100) - Module 1 (SAFETY)_96 RxPDO <-> Module 1 (SAFETY)/SAFETY FSoE Connection 1 Send Message/Message_4
//   Device 1 (EtherCAT) <-> Device 8 (EtherCAT)/Box 40 (AT5100-0100)
//     Term 1 (EK1200)/Term 13 (EL2912)/ConnectionInputs/TwinSafeGroup1.Box 40 (AT5100-0100) - Module 1 (SAFETY)_97 TxPDO <-> Module 1 (SAFETY)/SAFETY FSoE Connection 1 Receive Message/Message_4
//     Term 1 (EK1200)/Term 13 (EL2912)/ConnectionOutputs/TwinSafeGroup1.Box 40 (AT5100-0100) - Module 1 (SAFETY)_97 RxPDO <-> Module 1 (SAFETY)/SAFETY FSoE Connection 1 Send Message/Message_4
//   Device 1 (EtherCAT) <-> Device 8 (EtherCAT)/Box 41 (AT5100-0100)
//     Term 1 (EK1200)/Term 13 (EL2912)/ConnectionInputs/TwinSafeGroup1.Box 41 (AT5100-0100) - Module 1 (SAFETY)_98 TxPDO <-> Module 1 (SAFETY)/SAFETY FSoE Connection 1 Receive Message/Message_4
//     Term 1 (EK1200)/Term 13 (EL2912)/ConnectionOutputs/TwinSafeGroup1.Box 41 (AT5100-0100) - Module 1 (SAFETY)_98 RxPDO <-> Module 1 (SAFETY)/SAFETY FSoE Connection 1 Send Message/Message_4
//   Device 1 (EtherCAT) <-> Device 8 (EtherCAT)/Box 42 (AT5100-0100)
//     Term 1 (EK1200)/Term 13 (EL2912)/ConnectionInputs/TwinSafeGroup1.Box 42 (AT5100-0100) - Module 1 (SAFETY)_99 TxPDO <-> Module 1 (SAFETY)/SAFETY FSoE Connection 1 Receive Message/Message_4
//     Term 1 (EK1200)/Term 13 (EL2912)/ConnectionOutputs/TwinSafeGroup1.Box 42 (AT5100-0100) - Module 1 (SAFETY)_99 RxPDO <-> Module 1 (SAFETY)/SAFETY FSoE Connection 1 Send Message/Message_4
//   Device 1 (EtherCAT) <-> Device 8 (EtherCAT)/Box 43 (AT5100-0100)
//     Term 1 (EK1200)/Term 13 (EL2912)/ConnectionInputs/TwinSafeGroup1.Box 43 (AT5100-0100) - Module 1 (SAFETY)_100 TxPDO <-> Module 1 (SAFETY)/SAFETY FSoE Connection 1 Receive Message/Message_4
//     Term 1 (EK1200)/Term 13 (EL2912)/ConnectionOutputs/TwinSafeGroup1.Box 43 (AT5100-0100) - Module 1 (SAFETY)_100 RxPDO <-> Module 1 (SAFETY)/SAFETY FSoE Connection 1 Send Message/Message_4
//   Device 1 (EtherCAT) <-> Device 8 (EtherCAT)/Box 44 (AT5100-0100)
//     Term 1 (EK1200)/Term 13 (EL2912)/ConnectionInputs/TwinSafeGroup1.Box 44 (AT5100-0100) - Module 1 (SAFETY)_101 TxPDO <-> Module 1 (SAFETY)/SAFETY FSoE Connection 1 Receive Message/Message_4
//     Term 1 (EK1200)/Term 13 (EL2912)/ConnectionOutputs/TwinSafeGroup1.Box 44 (AT5100-0100) - Module 1 (SAFETY)_101 RxPDO <-> Module 1 (SAFETY)/SAFETY FSoE Connection 1 Send Message/Message_4
//   Device 1 (EtherCAT) <-> Device 8 (EtherCAT)/Box 45 (AT5100-0100)
//     Term 1 (EK1200)/Term 13 (EL2912)/ConnectionInputs/TwinSafeGroup1.Box 45 (AT5100-0100) - Module 1 (SAFETY)_102 TxPDO <-> Module 1 (SAFETY)/SAFETY FSoE Connection 1 Receive Message/Message_4
//   Device 1 (EtherCAT) <-> Device 8 (EtherCAT)/Box 46 (AT5100-0100)
//     Term 1 (EK1200)/Term 13 (EL2912)/ConnectionInputs/TwinSafeGroup1.Box 46 (AT5100-0100) - Module 1 (SAFETY)_103 TxPDO <-> Module 1 (SAFETY)/SAFETY FSoE Connection 1 Receive Message/Message_4
//     Term 1 (EK1200)/Term 13 (EL2912)/ConnectionOutputs/TwinSafeGroup1.Box 46 (AT5100-0100) - Module 1 (SAFETY)_103 RxPDO <-> Module 1 (SAFETY)/SAFETY FSoE Connection 1 Send Message/Message_4
//   Device 1 (EtherCAT) <-> Device 8 (EtherCAT)/Box 47 (AT5100-0100)
//     Term 1 (EK1200)/Term 13 (EL2912)/ConnectionInputs/TwinSafeGroup1.Box 47 (AT5100-0100) - Module 1 (SAFETY)_104 TxPDO <-> Module 1 (SAFETY)/SAFETY FSoE Connection 1 Receive Message/Message_4
//     Term 1 (EK1200)/Term 13 (EL2912)/ConnectionOutputs/TwinSafeGroup1.Box 47 (AT5100-0100) - Module 1 (SAFETY)_104 RxPDO <-> Module 1 (SAFETY)/SAFETY FSoE Connection 1 Send Message/Message_4
//   Device 1 (EtherCAT) <-> Device 8 (EtherCAT)/Box 48 (AT5100-0100)
//     Term 1 (EK1200)/Term 13 (EL2912)/ConnectionInputs/TwinSafeGroup1.Box 48 (AT5100-0100) - Module 1 (SAFETY)_105 TxPDO <-> Module 1 (SAFETY)/SAFETY FSoE Connection 1 Receive Message/Message_4
//     Term 1 (EK1200)/Term 13 (EL2912)/ConnectionOutputs/TwinSafeGroup1.Box 48 (AT5100-0100) - Module 1 (SAFETY)_105 RxPDO <-> Module 1 (SAFETY)/SAFETY FSoE Connection 1 Send Message/Message_4
//   Device 1 (EtherCAT) <-> Device 8 (EtherCAT)/Box 49 (AT5100-0100)
//     Term 1 (EK1200)/Term 13 (EL2912)/ConnectionInputs/TwinSafeGroup1.Box 49 (AT5100-0100) - Module 1 (SAFETY)_106 TxPDO <-> Module 1 (SAFETY)/SAFETY FSoE Connection 1 Receive Message/Message_4
//     Term 1 (EK1200)/Term 13 (EL2912)/ConnectionOutputs/TwinSafeGroup1.Box 49 (AT5100-0100) - Module 1 (SAFETY)_106 RxPDO <-> Module 1 (SAFETY)/SAFETY FSoE Connection 1 Send Message/Message_4
//   Device 4 (EtherCAT) <-> Device 1 (EtherCAT)/Term 1 (EK1200)/Term 13 (EL2912)
//     Box 59 (AT5100-0100)/Module 1 (SAFETY)/SAFETY FSoE Connection 1 Receive Message/Message_4 <-> ConnectionInputs/TwinSafeGroup1.Box 59 (AT5100-0100) - Module 1 (SAFETY)_116 TxPDO
//     Box 74 (AT5100-0100)/Module 1 (SAFETY)/SAFETY FSoE Connection 1 Receive Message/Message_4 <-> ConnectionInputs/TwinSafeGroup1.Box 74 (AT5100-0100) - Module 1 (SAFETY)_131 TxPDO
//     Box 61 (AT5100-0100)/Module 1 (SAFETY)/SAFETY FSoE Connection 1 Send Message/Message_4 <-> ConnectionOutputs/TwinSafeGroup1.Box 61 (AT5100-0100) - Module 1 (SAFETY)_118 RxPDO
//     Box 62 (AT5100-0100)/Module 1 (SAFETY)/SAFETY FSoE Connection 1 Send Message/Message_4 <-> ConnectionOutputs/TwinSafeGroup1.Box 62 (AT5100-0100) - Module 1 (SAFETY)_119 RxPDO
//   Device 4 (EtherCAT) <-> TcCOM Objects/XTS ProcessingUnit 1/XL Part 1/XL Module 34
//     Box 50 (AT5100-0100)/DRV Commutation angle/Commutation angle <-> Data Pointer/CommutationAngle
//     Box 50 (AT5100-0100)/DRV Controlword/Controlword <-> Data Pointer/Control
//     Box 50 (AT5100-0100)/DRV Statusword/Statusword <-> Data Pointer/Status
//     Box 50 (AT5100-0100)/DRV Target torque/Target torque <-> Data Pointer/Torque
//     Box 50 (AT5100-0100)/XFB Inputs/Data <-> Data Pointer/HallSensorValues
//   Device 4 (EtherCAT) <-> TcCOM Objects/XTS ProcessingUnit 1/XL Part 1/XL Module 35
//     Box 51 (AT5100-0100)/DRV Commutation angle/Commutation angle <-> Data Pointer/CommutationAngle
//     Box 51 (AT5100-0100)/DRV Controlword/Controlword <-> Data Pointer/Control
//     Box 51 (AT5100-0100)/DRV Statusword/Statusword <-> Data Pointer/Status
//     Box 51 (AT5100-0100)/DRV Target torque/Target torque <-> Data Pointer/Torque
//     Box 51 (AT5100-0100)/XFB Inputs/Data <-> Data Pointer/HallSensorValues
//   Device 4 (EtherCAT) <-> TcCOM Objects/XTS ProcessingUnit 1/XL Part 1/XL Module 36
//     Box 52 (AT5100-0100)/DRV Commutation angle/Commutation angle <-> Data Pointer/CommutationAngle
//     Box 52 (AT5100-0100)/DRV Controlword/Controlword <-> Data Pointer/Control
//     Box 52 (AT5100-0100)/DRV Statusword/Statusword <-> Data Pointer/Status
//     Box 52 (AT5100-0100)/DRV Target torque/Target torque <-> Data Pointer/Torque
//     Box 52 (AT5100-0100)/XFB Inputs/Data <-> Data Pointer/HallSensorValues
//   Device 4 (EtherCAT) <-> TcCOM Objects/XTS ProcessingUnit 1/XL Part 1/XL Module 37
//     Box 53 (AT5100-0100)/DRV Commutation angle/Commutation angle <-> Data Pointer/CommutationAngle
//     Box 53 (AT5100-0100)/DRV Controlword/Controlword <-> Data Pointer/Control
//     Box 53 (AT5100-0100)/DRV Statusword/Statusword <-> Data Pointer/Status
//     Box 53 (AT5100-0100)/DRV Target torque/Target torque <-> Data Pointer/Torque
//     Box 53 (AT5100-0100)/XFB Inputs/Data <-> Data Pointer/HallSensorValues
//   Device 4 (EtherCAT) <-> TcCOM Objects/XTS ProcessingUnit 1/XL Part 1/XL Module 38
//     Box 54 (AT5100-0100)/DRV Commutation angle/Commutation angle <-> Data Pointer/CommutationAngle
//     Box 54 (AT5100-0100)/DRV Controlword/Controlword <-> Data Pointer/Control
//     Box 54 (AT5100-0100)/DRV Statusword/Statusword <-> Data Pointer/Status
//     Box 54 (AT5100-0100)/DRV Target torque/Target torque <-> Data Pointer/Torque
//     Box 54 (AT5100-0100)/XFB Inputs/Data <-> Data Pointer/HallSensorValues
//   Device 4 (EtherCAT) <-> TcCOM Objects/XTS ProcessingUnit 1/XL Part 1/XL Module 39
//     Box 55 (AT5100-0100)/DRV Commutation angle/Commutation angle <-> Data Pointer/CommutationAngle
//     Box 55 (AT5100-0100)/DRV Controlword/Controlword <-> Data Pointer/Control
//     Box 55 (AT5100-0100)/DRV Statusword/Statusword <-> Data Pointer/Status
//     Box 55 (AT5100-0100)/DRV Target torque/Target torque <-> Data Pointer/Torque
//     Box 55 (AT5100-0100)/XFB Inputs/Data <-> Data Pointer/HallSensorValues
//   Device 4 (EtherCAT) <-> TcCOM Objects/XTS ProcessingUnit 1/XL Part 1/XL Module 40
//     Box 56 (AT5100-0100)/DRV Commutation angle/Commutation angle <-> Data Pointer/CommutationAngle
//     Box 56 (AT5100-0100)/DRV Controlword/Controlword <-> Data Pointer/Control
//     Box 56 (AT5100-0100)/DRV Statusword/Statusword <-> Data Pointer/Status
//     Box 56 (AT5100-0100)/DRV Target torque/Target torque <-> Data Pointer/Torque
//     Box 56 (AT5100-0100)/XFB Inputs/Data <-> Data Pointer/HallSensorValues
//   Device 4 (EtherCAT) <-> TcCOM Objects/XTS ProcessingUnit 1/XL Part 1/XL Module 41
//     Box 57 (AT5100-0100)/DRV Commutation angle/Commutation angle <-> Data Pointer/CommutationAngle
//     Box 57 (AT5100-0100)/DRV Controlword/Controlword <-> Data Pointer/Control
//     Box 57 (AT5100-0100)/DRV Statusword/Statusword <-> Data Pointer/Status
//     Box 57 (AT5100-0100)/DRV Target torque/Target torque <-> Data Pointer/Torque
//     Box 57 (AT5100-0100)/XFB Inputs/Data <-> Data Pointer/HallSensorValues
//   Device 4 (EtherCAT) <-> TcCOM Objects/XTS ProcessingUnit 1/XL Part 1/XL Module 42
//     Box 58 (AT5100-0100)/DRV Commutation angle/Commutation angle <-> Data Pointer/CommutationAngle
//     Box 58 (AT5100-0100)/DRV Controlword/Controlword <-> Data Pointer/Control
//     Box 58 (AT5100-0100)/DRV Statusword/Statusword <-> Data Pointer/Status
//     Box 58 (AT5100-0100)/DRV Target torque/Target torque <-> Data Pointer/Torque
//     Box 58 (AT5100-0100)/XFB Inputs/Data <-> Data Pointer/HallSensorValues
//   Device 4 (EtherCAT) <-> TcCOM Objects/XTS ProcessingUnit 1/XL Part 1/XL Module 43
//     Box 59 (AT5100-0100)/DRV Commutation angle/Commutation angle <-> Data Pointer/CommutationAngle
//     Box 59 (AT5100-0100)/DRV Controlword/Controlword <-> Data Pointer/Control
//     Box 59 (AT5100-0100)/DRV Statusword/Statusword <-> Data Pointer/Status
//     Box 59 (AT5100-0100)/DRV Target torque/Target torque <-> Data Pointer/Torque
//     Box 59 (AT5100-0100)/XFB Inputs/Data <-> Data Pointer/HallSensorValues
//   Device 4 (EtherCAT) <-> TcCOM Objects/XTS ProcessingUnit 1/XL Part 1/XL Module 44
//     Box 60 (AT5100-0100)/DRV Commutation angle/Commutation angle <-> Data Pointer/CommutationAngle
//     Box 60 (AT5100-0100)/DRV Controlword/Controlword <-> Data Pointer/Control
//     Box 60 (AT5100-0100)/DRV Statusword/Statusword <-> Data Pointer/Status
//     Box 60 (AT5100-0100)/DRV Target torque/Target torque <-> Data Pointer/Torque
//     Box 60 (AT5100-0100)/XFB Inputs/Data <-> Data Pointer/HallSensorValues
//   Device 4 (EtherCAT) <-> TcCOM Objects/XTS ProcessingUnit 1/XL Part 1/XL Module 45
//     Box 61 (AT5100-0100)/DRV Commutation angle/Commutation angle <-> Data Pointer/CommutationAngle
//     Box 61 (AT5100-0100)/DRV Controlword/Controlword <-> Data Pointer/Control
//     Box 61 (AT5100-0100)/DRV Statusword/Statusword <-> Data Pointer/Status
//     Box 61 (AT5100-0100)/DRV Target torque/Target torque <-> Data Pointer/Torque
//     Box 61 (AT5100-0100)/XFB Inputs/Data <-> Data Pointer/HallSensorValues
//   Device 4 (EtherCAT) <-> TcCOM Objects/XTS ProcessingUnit 1/XL Part 2/XL Module 48
//     Box 70 (AT5100-0100)/DRV Commutation angle/Commutation angle <-> Data Pointer/CommutationAngle
//     Box 70 (AT5100-0100)/DRV Controlword/Controlword <-> Data Pointer/Control
//     Box 70 (AT5100-0100)/DRV Statusword/Statusword <-> Data Pointer/Status
//     Box 70 (AT5100-0100)/DRV Target torque/Target torque <-> Data Pointer/Torque
//     Box 70 (AT5100-0100)/XFB Inputs/Data <-> Data Pointer/HallSensorValues
//   Device 4 (EtherCAT) <-> TcCOM Objects/XTS ProcessingUnit 1/XL Part 2/XL Module 49
//     Box 71 (AT5100-0100)/DRV Commutation angle/Commutation angle <-> Data Pointer/CommutationAngle
//     Box 71 (AT5100-0100)/DRV Controlword/Controlword <-> Data Pointer/Control
//     Box 71 (AT5100-0100)/DRV Statusword/Statusword <-> Data Pointer/Status
//     Box 71 (AT5100-0100)/DRV Target torque/Target torque <-> Data Pointer/Torque
//     Box 71 (AT5100-0100)/XFB Inputs/Data <-> Data Pointer/HallSensorValues
//   Device 4 (EtherCAT) <-> TcCOM Objects/XTS ProcessingUnit 1/XL Part 2/XL Module 50
//     Box 62 (AT5100-0100)/DRV Commutation angle/Commutation angle <-> Data Pointer/CommutationAngle
//     Box 62 (AT5100-0100)/DRV Controlword/Controlword <-> Data Pointer/Control
//     Box 62 (AT5100-0100)/DRV Statusword/Statusword <-> Data Pointer/Status
//     Box 62 (AT5100-0100)/DRV Target torque/Target torque <-> Data Pointer/Torque
//     Box 62 (AT5100-0100)/XFB Inputs/Data <-> Data Pointer/HallSensorValues
//   Device 4 (EtherCAT) <-> TcCOM Objects/XTS ProcessingUnit 1/XL Part 2/XL Module 51
//     Box 63 (AT5100-0100)/DRV Commutation angle/Commutation angle <-> Data Pointer/CommutationAngle
//     Box 63 (AT5100-0100)/DRV Controlword/Controlword <-> Data Pointer/Control
//     Box 63 (AT5100-0100)/DRV Statusword/Statusword <-> Data Pointer/Status
//     Box 63 (AT5100-0100)/DRV Target torque/Target torque <-> Data Pointer/Torque
//     Box 63 (AT5100-0100)/XFB Inputs/Data <-> Data Pointer/HallSensorValues
//   Device 4 (EtherCAT) <-> TcCOM Objects/XTS ProcessingUnit 1/XL Part 2/XL Module 52
//     Box 64 (AT5100-0100)/DRV Commutation angle/Commutation angle <-> Data Pointer/CommutationAngle
//     Box 64 (AT5100-0100)/DRV Controlword/Controlword <-> Data Pointer/Control
//     Box 64 (AT5100-0100)/DRV Statusword/Statusword <-> Data Pointer/Status
//     Box 64 (AT5100-0100)/DRV Target torque/Target torque <-> Data Pointer/Torque
//     Box 64 (AT5100-0100)/XFB Inputs/Data <-> Data Pointer/HallSensorValues
//   Device 4 (EtherCAT) <-> TcCOM Objects/XTS ProcessingUnit 1/XL Part 2/XL Module 53
//     Box 65 (AT5100-0100)/DRV Commutation angle/Commutation angle <-> Data Pointer/CommutationAngle
//     Box 65 (AT5100-0100)/DRV Controlword/Controlword <-> Data Pointer/Control
//     Box 65 (AT5100-0100)/DRV Statusword/Statusword <-> Data Pointer/Status
//     Box 65 (AT5100-0100)/DRV Target torque/Target torque <-> Data Pointer/Torque
//     Box 65 (AT5100-0100)/XFB Inputs/Data <-> Data Pointer/HallSensorValues
//   Device 4 (EtherCAT) <-> TcCOM Objects/XTS ProcessingUnit 1/XL Part 2/XL Module 54
//     Box 66 (AT5100-0100)/DRV Commutation angle/Commutation angle <-> Data Pointer/CommutationAngle
//     Box 66 (AT5100-0100)/DRV Controlword/Controlword <-> Data Pointer/Control
//     Box 66 (AT5100-0100)/DRV Statusword/Statusword <-> Data Pointer/Status
//     Box 66 (AT5100-0100)/DRV Target torque/Target torque <-> Data Pointer/Torque
//     Box 66 (AT5100-0100)/XFB Inputs/Data <-> Data Pointer/HallSensorValues
//   Device 4 (EtherCAT) <-> TcCOM Objects/XTS ProcessingUnit 1/XL Part 2/XL Module 55
//     Box 67 (AT5100-0100)/DRV Commutation angle/Commutation angle <-> Data Pointer/CommutationAngle
//     Box 67 (AT5100-0100)/DRV Controlword/Controlword <-> Data Pointer/Control
//     Box 67 (AT5100-0100)/DRV Statusword/Statusword <-> Data Pointer/Status
//     Box 67 (AT5100-0100)/DRV Target torque/Target torque <-> Data Pointer/Torque
//     Box 67 (AT5100-0100)/XFB Inputs/Data <-> Data Pointer/HallSensorValues
//   Device 4 (EtherCAT) <-> TcCOM Objects/XTS ProcessingUnit 1/XL Part 2/XL Module 56
//     Box 68 (AT5100-0100)/DRV Commutation angle/Commutation angle <-> Data Pointer/CommutationAngle
//     Box 68 (AT5100-0100)/DRV Controlword/Controlword <-> Data Pointer/Control
//     Box 68 (AT5100-0100)/DRV Statusword/Statusword <-> Data Pointer/Status
//     Box 68 (AT5100-0100)/DRV Target torque/Target torque <-> Data Pointer/Torque
//     Box 68 (AT5100-0100)/XFB Inputs/Data <-> Data Pointer/HallSensorValues
//   Device 4 (EtherCAT) <-> TcCOM Objects/XTS ProcessingUnit 1/XL Part 2/XL Module 57
//     Box 69 (AT5100-0100)/DRV Commutation angle/Commutation angle <-> Data Pointer/CommutationAngle
//     Box 69 (AT5100-0100)/DRV Controlword/Controlword <-> Data Pointer/Control
//     Box 69 (AT5100-0100)/DRV Statusword/Statusword <-> Data Pointer/Status
//     Box 69 (AT5100-0100)/DRV Target torque/Target torque <-> Data Pointer/Torque
//     Box 69 (AT5100-0100)/XFB Inputs/Data <-> Data Pointer/HallSensorValues
//   Device 4 (EtherCAT) <-> TcCOM Objects/XTS ProcessingUnit 1/XL Part 3/XL Module 1
//     Box 74 (AT5100-0100)/DRV Commutation angle/Commutation angle <-> Data Pointer/CommutationAngle
//     Box 74 (AT5100-0100)/DRV Controlword/Controlword <-> Data Pointer/Control
//     Box 74 (AT5100-0100)/DRV Statusword/Statusword <-> Data Pointer/Status
//     Box 74 (AT5100-0100)/DRV Target torque/Target torque <-> Data Pointer/Torque
//     Box 74 (AT5100-0100)/XFB Inputs/Data <-> Data Pointer/HallSensorValues
//   Device 4 (EtherCAT) <-> TcCOM Objects/XTS ProcessingUnit 1/XL Part 3/XL Module 2
//     Box 75 (AT5100-0100)/DRV Commutation angle/Commutation angle <-> Data Pointer/CommutationAngle
//     Box 75 (AT5100-0100)/DRV Controlword/Controlword <-> Data Pointer/Control
//     Box 75 (AT5100-0100)/DRV Statusword/Statusword <-> Data Pointer/Status
//     Box 75 (AT5100-0100)/DRV Target torque/Target torque <-> Data Pointer/Torque
//     Box 75 (AT5100-0100)/XFB Inputs/Data <-> Data Pointer/HallSensorValues
//   Device 4 (EtherCAT) <-> TcCOM Objects/XTS ProcessingUnit 1/XL Part 3/XL Module 3
//     Box 76 (AT5100-0100)/DRV Commutation angle/Commutation angle <-> Data Pointer/CommutationAngle
//     Box 76 (AT5100-0100)/DRV Controlword/Controlword <-> Data Pointer/Control
//     Box 76 (AT5100-0100)/DRV Statusword/Statusword <-> Data Pointer/Status
//     Box 76 (AT5100-0100)/DRV Target torque/Target torque <-> Data Pointer/Torque
//     Box 76 (AT5100-0100)/XFB Inputs/Data <-> Data Pointer/HallSensorValues
//   Device 4 (EtherCAT) <-> TcCOM Objects/XTS ProcessingUnit 1/XL Part 3/XL Module 4
//     Box 77 (AT5100-0100)/DRV Commutation angle/Commutation angle <-> Data Pointer/CommutationAngle
//     Box 77 (AT5100-0100)/DRV Controlword/Controlword <-> Data Pointer/Control
//     Box 77 (AT5100-0100)/DRV Statusword/Statusword <-> Data Pointer/Status
//     Box 77 (AT5100-0100)/DRV Target torque/Target torque <-> Data Pointer/Torque
//     Box 77 (AT5100-0100)/XFB Inputs/Data <-> Data Pointer/HallSensorValues
//   Device 4 (EtherCAT) <-> TcCOM Objects/XTS ProcessingUnit 1/XL Part 3/XL Module 46
//     Box 72 (AT5100-0100)/DRV Commutation angle/Commutation angle <-> Data Pointer/CommutationAngle
//     Box 72 (AT5100-0100)/DRV Controlword/Controlword <-> Data Pointer/Control
//     Box 72 (AT5100-0100)/DRV Statusword/Statusword <-> Data Pointer/Status
//     Box 72 (AT5100-0100)/DRV Target torque/Target torque <-> Data Pointer/Torque
//     Box 72 (AT5100-0100)/XFB Inputs/Data <-> Data Pointer/HallSensorValues
//   Device 4 (EtherCAT) <-> TcCOM Objects/XTS ProcessingUnit 1/XL Part 3/XL Module 47
//     Box 73 (AT5100-0100)/DRV Commutation angle/Commutation angle <-> Data Pointer/CommutationAngle
//     Box 73 (AT5100-0100)/DRV Controlword/Controlword <-> Data Pointer/Control
//     Box 73 (AT5100-0100)/DRV Statusword/Statusword <-> Data Pointer/Status
//     Box 73 (AT5100-0100)/DRV Target torque/Target torque <-> Data Pointer/Torque
//     Box 73 (AT5100-0100)/XFB Inputs/Data <-> Data Pointer/HallSensorValues
//   Device 4 (EtherCAT) <-> TcCOM Objects/XTS ProcessingUnit 1/XL Part 3/XL Module 5
//     Box 78 (AT5100-0100)/DRV Commutation angle/Commutation angle <-> Data Pointer/CommutationAngle
//     Box 78 (AT5100-0100)/DRV Controlword/Controlword <-> Data Pointer/Control
//     Box 78 (AT5100-0100)/DRV Statusword/Statusword <-> Data Pointer/Status
//     Box 78 (AT5100-0100)/DRV Target torque/Target torque <-> Data Pointer/Torque
//     Box 78 (AT5100-0100)/XFB Inputs/Data <-> Data Pointer/HallSensorValues
//   Device 4 (EtherCAT) <-> TcCOM Objects/XTS ProcessingUnit 1/XL Part 3/XL Module 6
//     Box 79 (AT5100-0100)/DRV Commutation angle/Commutation angle <-> Data Pointer/CommutationAngle
//     Box 79 (AT5100-0100)/DRV Controlword/Controlword <-> Data Pointer/Control
//     Box 79 (AT5100-0100)/DRV Statusword/Statusword <-> Data Pointer/Status
//     Box 79 (AT5100-0100)/DRV Target torque/Target torque <-> Data Pointer/Torque
//     Box 79 (AT5100-0100)/XFB Inputs/Data <-> Data Pointer/HallSensorValues
//   Device 4 (EtherCAT) <-> TcCOM Objects/XTS ProcessingUnit 1/XL Part 3/XL Module 7
//     Box 80 (AT5100-0100)/DRV Commutation angle/Commutation angle <-> Data Pointer/CommutationAngle
//     Box 80 (AT5100-0100)/DRV Controlword/Controlword <-> Data Pointer/Control
//     Box 80 (AT5100-0100)/DRV Statusword/Statusword <-> Data Pointer/Status
//     Box 80 (AT5100-0100)/DRV Target torque/Target torque <-> Data Pointer/Torque
//     Box 80 (AT5100-0100)/XFB Inputs/Data <-> Data Pointer/HallSensorValues
//   Device 4 (EtherCAT) <-> TcCOM Objects/XTS ProcessingUnit 1/XL Part 3/XL Module 8
//     Box 81 (AT5100-0100)/DRV Commutation angle/Commutation angle <-> Data Pointer/CommutationAngle
//     Box 81 (AT5100-0100)/DRV Controlword/Controlword <-> Data Pointer/Control
//     Box 81 (AT5100-0100)/DRV Statusword/Statusword <-> Data Pointer/Status
//     Box 81 (AT5100-0100)/DRV Target torque/Target torque <-> Data Pointer/Torque
//     Box 81 (AT5100-0100)/XFB Inputs/Data <-> Data Pointer/HallSensorValues
//   Device 8 (EtherCAT) <-> Device 1 (EtherCAT)/Term 1 (EK1200)/Term 13 (EL2912)
//     Box 24 (AT5100-0100)/Module 1 (SAFETY)/SAFETY FSoE Connection 1 Receive Message/Message_4 <-> ConnectionInputs/TwinSafeGroup1.Box 24 (AT5100-0100) - Module 1 (SAFETY)_81 TxPDO
//     Box 45 (AT5100-0100)/Module 1 (SAFETY)/SAFETY FSoE Connection 1 Send Message/Message_4 <-> ConnectionOutputs/TwinSafeGroup1.Box 45 (AT5100-0100) - Module 1 (SAFETY)_102 RxPDO
//   Device 8 (EtherCAT) <-> TcCOM Objects/XTS ProcessingUnit 1/XL Part 1/XL Module 19
//     Box 38 (AT5100-0100)/DRV Commutation angle/Commutation angle <-> Data Pointer/CommutationAngle
//     Box 38 (AT5100-0100)/DRV Controlword/Controlword <-> Data Pointer/Control
//     Box 38 (AT5100-0100)/DRV Statusword/Statusword <-> Data Pointer/Status
//     Box 38 (AT5100-0100)/DRV Target torque/Target torque <-> Data Pointer/Torque
//     Box 38 (AT5100-0100)/XFB Inputs/Data <-> Data Pointer/HallSensorValues
//   Device 8 (EtherCAT) <-> TcCOM Objects/XTS ProcessingUnit 1/XL Part 1/XL Module 20
//     Box 39 (AT5100-0100)/DRV Commutation angle/Commutation angle <-> Data Pointer/CommutationAngle
//     Box 39 (AT5100-0100)/DRV Controlword/Controlword <-> Data Pointer/Control
//     Box 39 (AT5100-0100)/DRV Statusword/Statusword <-> Data Pointer/Status
//     Box 39 (AT5100-0100)/DRV Target torque/Target torque <-> Data Pointer/Torque
//     Box 39 (AT5100-0100)/XFB Inputs/Data <-> Data Pointer/HallSensorValues
//   Device 8 (EtherCAT) <-> TcCOM Objects/XTS ProcessingUnit 1/XL Part 1/XL Module 21
//     Box 40 (AT5100-0100)/DRV Commutation angle/Commutation angle <-> Data Pointer/CommutationAngle
//     Box 40 (AT5100-0100)/DRV Controlword/Controlword <-> Data Pointer/Control
//     Box 40 (AT5100-0100)/DRV Statusword/Statusword <-> Data Pointer/Status
//     Box 40 (AT5100-0100)/DRV Target torque/Target torque <-> Data Pointer/Torque
//     Box 40 (AT5100-0100)/XFB Inputs/Data <-> Data Pointer/HallSensorValues
//   Device 8 (EtherCAT) <-> TcCOM Objects/XTS ProcessingUnit 1/XL Part 1/XL Module 22
//     Box 41 (AT5100-0100)/DRV Commutation angle/Commutation angle <-> Data Pointer/CommutationAngle
//     Box 41 (AT5100-0100)/DRV Controlword/Controlword <-> Data Pointer/Control
//     Box 41 (AT5100-0100)/DRV Statusword/Statusword <-> Data Pointer/Status
//     Box 41 (AT5100-0100)/DRV Target torque/Target torque <-> Data Pointer/Torque
//     Box 41 (AT5100-0100)/XFB Inputs/Data <-> Data Pointer/HallSensorValues
//   Device 8 (EtherCAT) <-> TcCOM Objects/XTS ProcessingUnit 1/XL Part 1/XL Module 26
//     Box 42 (AT5100-0100)/DRV Commutation angle/Commutation angle <-> Data Pointer/CommutationAngle
//     Box 42 (AT5100-0100)/DRV Controlword/Controlword <-> Data Pointer/Control
//     Box 42 (AT5100-0100)/DRV Statusword/Statusword <-> Data Pointer/Status
//     Box 42 (AT5100-0100)/DRV Target torque/Target torque <-> Data Pointer/Torque
//     Box 42 (AT5100-0100)/XFB Inputs/Data <-> Data Pointer/HallSensorValues
//   Device 8 (EtherCAT) <-> TcCOM Objects/XTS ProcessingUnit 1/XL Part 1/XL Module 27
//     Box 43 (AT5100-0100)/DRV Commutation angle/Commutation angle <-> Data Pointer/CommutationAngle
//     Box 43 (AT5100-0100)/DRV Controlword/Controlword <-> Data Pointer/Control
//     Box 43 (AT5100-0100)/DRV Statusword/Statusword <-> Data Pointer/Status
//     Box 43 (AT5100-0100)/DRV Target torque/Target torque <-> Data Pointer/Torque
//     Box 43 (AT5100-0100)/XFB Inputs/Data <-> Data Pointer/HallSensorValues
//   Device 8 (EtherCAT) <-> TcCOM Objects/XTS ProcessingUnit 1/XL Part 1/XL Module 28
//     Box 44 (AT5100-0100)/DRV Commutation angle/Commutation angle <-> Data Pointer/CommutationAngle
//     Box 44 (AT5100-0100)/DRV Controlword/Controlword <-> Data Pointer/Control
//     Box 44 (AT5100-0100)/DRV Statusword/Statusword <-> Data Pointer/Status
//     Box 44 (AT5100-0100)/DRV Target torque/Target torque <-> Data Pointer/Torque
//     Box 44 (AT5100-0100)/XFB Inputs/Data <-> Data Pointer/HallSensorValues
//   Device 8 (EtherCAT) <-> TcCOM Objects/XTS ProcessingUnit 1/XL Part 1/XL Module 29
//     Box 45 (AT5100-0100)/DRV Commutation angle/Commutation angle <-> Data Pointer/CommutationAngle
//     Box 45 (AT5100-0100)/DRV Controlword/Controlword <-> Data Pointer/Control
//     Box 45 (AT5100-0100)/DRV Statusword/Statusword <-> Data Pointer/Status
//     Box 45 (AT5100-0100)/DRV Target torque/Target torque <-> Data Pointer/Torque
//     Box 45 (AT5100-0100)/XFB Inputs/Data <-> Data Pointer/HallSensorValues
//   Device 8 (EtherCAT) <-> TcCOM Objects/XTS ProcessingUnit 1/XL Part 1/XL Module 30
//     Box 46 (AT5100-0100)/DRV Commutation angle/Commutation angle <-> Data Pointer/CommutationAngle
//     Box 46 (AT5100-0100)/DRV Controlword/Controlword <-> Data Pointer/Control
//     Box 46 (AT5100-0100)/DRV Statusword/Statusword <-> Data Pointer/Status
//     Box 46 (AT5100-0100)/DRV Target torque/Target torque <-> Data Pointer/Torque
//     Box 46 (AT5100-0100)/XFB Inputs/Data <-> Data Pointer/HallSensorValues
//   Device 8 (EtherCAT) <-> TcCOM Objects/XTS ProcessingUnit 1/XL Part 1/XL Module 31
//     Box 47 (AT5100-0100)/DRV Commutation angle/Commutation angle <-> Data Pointer/CommutationAngle
//     Box 47 (AT5100-0100)/DRV Controlword/Controlword <-> Data Pointer/Control
//     Box 47 (AT5100-0100)/DRV Statusword/Statusword <-> Data Pointer/Status
//     Box 47 (AT5100-0100)/DRV Target torque/Target torque <-> Data Pointer/Torque
//     Box 47 (AT5100-0100)/XFB Inputs/Data <-> Data Pointer/HallSensorValues
//   Device 8 (EtherCAT) <-> TcCOM Objects/XTS ProcessingUnit 1/XL Part 1/XL Module 32
//     Box 48 (AT5100-0100)/DRV Commutation angle/Commutation angle <-> Data Pointer/CommutationAngle
//     Box 48 (AT5100-0100)/DRV Controlword/Controlword <-> Data Pointer/Control
//     Box 48 (AT5100-0100)/DRV Statusword/Statusword <-> Data Pointer/Status
//     Box 48 (AT5100-0100)/DRV Target torque/Target torque <-> Data Pointer/Torque
//     Box 48 (AT5100-0100)/XFB Inputs/Data <-> Data Pointer/HallSensorValues
//   Device 8 (EtherCAT) <-> TcCOM Objects/XTS ProcessingUnit 1/XL Part 1/XL Module 33
//     Box 49 (AT5100-0100)/DRV Commutation angle/Commutation angle <-> Data Pointer/CommutationAngle
//     Box 49 (AT5100-0100)/DRV Controlword/Controlword <-> Data Pointer/Control
//     Box 49 (AT5100-0100)/DRV Statusword/Statusword <-> Data Pointer/Status
//     Box 49 (AT5100-0100)/DRV Target torque/Target torque <-> Data Pointer/Torque
//     Box 49 (AT5100-0100)/XFB Inputs/Data <-> Data Pointer/HallSensorValues
//   Device 8 (EtherCAT) <-> TcCOM Objects/XTS ProcessingUnit 1/XL Part 2/XL Module 23
//     Box 37 (AT5100-0100)/DRV Commutation angle/Commutation angle <-> Data Pointer/CommutationAngle
//     Box 37 (AT5100-0100)/DRV Controlword/Controlword <-> Data Pointer/Control
//     Box 37 (AT5100-0100)/DRV Statusword/Statusword <-> Data Pointer/Status
//     Box 37 (AT5100-0100)/DRV Target torque/Target torque <-> Data Pointer/Torque
//     Box 37 (AT5100-0100)/XFB Inputs/Data <-> Data Pointer/HallSensorValues
//   Device 8 (EtherCAT) <-> TcCOM Objects/XTS ProcessingUnit 1/XL Part 2/XL Module 24
//     Box 28 (AT5100-0100)/DRV Commutation angle/Commutation angle <-> Data Pointer/CommutationAngle
//     Box 28 (AT5100-0100)/DRV Controlword/Controlword <-> Data Pointer/Control
//     Box 28 (AT5100-0100)/DRV Statusword/Statusword <-> Data Pointer/Status
//     Box 28 (AT5100-0100)/DRV Target torque/Target torque <-> Data Pointer/Torque
//     Box 28 (AT5100-0100)/XFB Inputs/Data <-> Data Pointer/HallSensorValues
//   Device 8 (EtherCAT) <-> TcCOM Objects/XTS ProcessingUnit 1/XL Part 2/XL Module 25
//     Box 29 (AT5100-0100)/DRV Commutation angle/Commutation angle <-> Data Pointer/CommutationAngle
//     Box 29 (AT5100-0100)/DRV Controlword/Controlword <-> Data Pointer/Control
//     Box 29 (AT5100-0100)/DRV Statusword/Statusword <-> Data Pointer/Status
//     Box 29 (AT5100-0100)/DRV Target torque/Target torque <-> Data Pointer/Torque
//     Box 29 (AT5100-0100)/XFB Inputs/Data <-> Data Pointer/HallSensorValues
//   Device 8 (EtherCAT) <-> TcCOM Objects/XTS ProcessingUnit 1/XL Part 2/XL Module 58
//     Box 30 (AT5100-0100)/DRV Commutation angle/Commutation angle <-> Data Pointer/CommutationAngle
//     Box 30 (AT5100-0100)/DRV Controlword/Controlword <-> Data Pointer/Control
//     Box 30 (AT5100-0100)/DRV Statusword/Statusword <-> Data Pointer/Status
//     Box 30 (AT5100-0100)/DRV Target torque/Target torque <-> Data Pointer/Torque
//     Box 30 (AT5100-0100)/XFB Inputs/Data <-> Data Pointer/HallSensorValues
//   Device 8 (EtherCAT) <-> TcCOM Objects/XTS ProcessingUnit 1/XL Part 2/XL Module 59
//     Box 31 (AT5100-0100)/DRV Commutation angle/Commutation angle <-> Data Pointer/CommutationAngle
//     Box 31 (AT5100-0100)/DRV Controlword/Controlword <-> Data Pointer/Control
//     Box 31 (AT5100-0100)/DRV Statusword/Statusword <-> Data Pointer/Status
//     Box 31 (AT5100-0100)/DRV Target torque/Target torque <-> Data Pointer/Torque
//     Box 31 (AT5100-0100)/XFB Inputs/Data <-> Data Pointer/HallSensorValues
//   Device 8 (EtherCAT) <-> TcCOM Objects/XTS ProcessingUnit 1/XL Part 2/XL Module 60
//     Box 32 (AT5100-0100)/DRV Commutation angle/Commutation angle <-> Data Pointer/CommutationAngle
//     Box 32 (AT5100-0100)/DRV Controlword/Controlword <-> Data Pointer/Control
//     Box 32 (AT5100-0100)/DRV Statusword/Statusword <-> Data Pointer/Status
//     Box 32 (AT5100-0100)/DRV Target torque/Target torque <-> Data Pointer/Torque
//     Box 32 (AT5100-0100)/XFB Inputs/Data <-> Data Pointer/HallSensorValues
//   Device 8 (EtherCAT) <-> TcCOM Objects/XTS ProcessingUnit 1/XL Part 2/XL Module 61
//     Box 33 (AT5100-0100)/DRV Commutation angle/Commutation angle <-> Data Pointer/CommutationAngle
//     Box 33 (AT5100-0100)/DRV Controlword/Controlword <-> Data Pointer/Control
//     Box 33 (AT5100-0100)/DRV Statusword/Statusword <-> Data Pointer/Status
//     Box 33 (AT5100-0100)/DRV Target torque/Target torque <-> Data Pointer/Torque
//     Box 33 (AT5100-0100)/XFB Inputs/Data <-> Data Pointer/HallSensorValues
//   Device 8 (EtherCAT) <-> TcCOM Objects/XTS ProcessingUnit 1/XL Part 2/XL Module 62
//     Box 34 (AT5100-0100)/DRV Commutation angle/Commutation angle <-> Data Pointer/CommutationAngle
//     Box 34 (AT5100-0100)/DRV Controlword/Controlword <-> Data Pointer/Control
//     Box 34 (AT5100-0100)/DRV Statusword/Statusword <-> Data Pointer/Status
//     Box 34 (AT5100-0100)/DRV Target torque/Target torque <-> Data Pointer/Torque
//     Box 34 (AT5100-0100)/XFB Inputs/Data <-> Data Pointer/HallSensorValues
//   Device 8 (EtherCAT) <-> TcCOM Objects/XTS ProcessingUnit 1/XL Part 2/XL Module 63
//     Box 35 (AT5100-0100)/DRV Commutation angle/Commutation angle <-> Data Pointer/CommutationAngle
//     Box 35 (AT5100-0100)/DRV Controlword/Controlword <-> Data Pointer/Control
//     Box 35 (AT5100-0100)/DRV Statusword/Statusword <-> Data Pointer/Status
//     Box 35 (AT5100-0100)/DRV Target torque/Target torque <-> Data Pointer/Torque
//     Box 35 (AT5100-0100)/XFB Inputs/Data <-> Data Pointer/HallSensorValues
//   Device 8 (EtherCAT) <-> TcCOM Objects/XTS ProcessingUnit 1/XL Part 2/XL Module 64
//     Box 36 (AT5100-0100)/DRV Commutation angle/Commutation angle <-> Data Pointer/CommutationAngle
//     Box 36 (AT5100-0100)/DRV Controlword/Controlword <-> Data Pointer/Control
//     Box 36 (AT5100-0100)/DRV Statusword/Statusword <-> Data Pointer/Status
//     Box 36 (AT5100-0100)/DRV Target torque/Target torque <-> Data Pointer/Torque
//     Box 36 (AT5100-0100)/XFB Inputs/Data <-> Data Pointer/HallSensorValues
//   Device 8 (EtherCAT) <-> TcCOM Objects/XTS ProcessingUnit 1/XL Part 3/XL Module 10
//     Box 19 (AT5100-0100)/DRV Commutation angle/Commutation angle <-> Data Pointer/CommutationAngle
//     Box 19 (AT5100-0100)/DRV Controlword/Controlword <-> Data Pointer/Control
//     Box 19 (AT5100-0100)/DRV Statusword/Statusword <-> Data Pointer/Status
//     Box 19 (AT5100-0100)/DRV Target torque/Target torque <-> Data Pointer/Torque
//     Box 19 (AT5100-0100)/XFB Inputs/Data <-> Data Pointer/HallSensorValues
//   Device 8 (EtherCAT) <-> TcCOM Objects/XTS ProcessingUnit 1/XL Part 3/XL Module 11
//     Box 20 (AT5100-0100)/DRV Commutation angle/Commutation angle <-> Data Pointer/CommutationAngle
//     Box 20 (AT5100-0100)/DRV Controlword/Controlword <-> Data Pointer/Control
//     Box 20 (AT5100-0100)/DRV Statusword/Statusword <-> Data Pointer/Status
//     Box 20 (AT5100-0100)/DRV Target torque/Target torque <-> Data Pointer/Torque
//     Box 20 (AT5100-0100)/XFB Inputs/Data <-> Data Pointer/HallSensorValues
//   Device 8 (EtherCAT) <-> TcCOM Objects/XTS ProcessingUnit 1/XL Part 3/XL Module 12
//     Box 21 (AT5100-0100)/DRV Commutation angle/Commutation angle <-> Data Pointer/CommutationAngle
//     Box 21 (AT5100-0100)/DRV Controlword/Controlword <-> Data Pointer/Control
//     Box 21 (AT5100-0100)/DRV Statusword/Statusword <-> Data Pointer/Status
//     Box 21 (AT5100-0100)/DRV Target torque/Target torque <-> Data Pointer/Torque
//     Box 21 (AT5100-0100)/XFB Inputs/Data <-> Data Pointer/HallSensorValues
//   Device 8 (EtherCAT) <-> TcCOM Objects/XTS ProcessingUnit 1/XL Part 3/XL Module 13
//     Box 22 (AT5100-0100)/DRV Commutation angle/Commutation angle <-> Data Pointer/CommutationAngle
//     Box 22 (AT5100-0100)/DRV Controlword/Controlword <-> Data Pointer/Control
//     Box 22 (AT5100-0100)/DRV Statusword/Statusword <-> Data Pointer/Status
//     Box 22 (AT5100-0100)/DRV Target torque/Target torque <-> Data Pointer/Torque
//     Box 22 (AT5100-0100)/XFB Inputs/Data <-> Data Pointer/HallSensorValues
//   Device 8 (EtherCAT) <-> TcCOM Objects/XTS ProcessingUnit 1/XL Part 3/XL Module 14
//     Box 23 (AT5100-0100)/DRV Commutation angle/Commutation angle <-> Data Pointer/CommutationAngle
//     Box 23 (AT5100-0100)/DRV Controlword/Controlword <-> Data Pointer/Control
//     Box 23 (AT5100-0100)/DRV Statusword/Statusword <-> Data Pointer/Status
//     Box 23 (AT5100-0100)/DRV Target torque/Target torque <-> Data Pointer/Torque
//     Box 23 (AT5100-0100)/XFB Inputs/Data <-> Data Pointer/HallSensorValues
//   Device 8 (EtherCAT) <-> TcCOM Objects/XTS ProcessingUnit 1/XL Part 3/XL Module 15
//     Box 24 (AT5100-0100)/DRV Commutation angle/Commutation angle <-> Data Pointer/CommutationAngle
//     Box 24 (AT5100-0100)/DRV Controlword/Controlword <-> Data Pointer/Control
//     Box 24 (AT5100-0100)/DRV Statusword/Statusword <-> Data Pointer/Status
//     Box 24 (AT5100-0100)/DRV Target torque/Target torque <-> Data Pointer/Torque
//     Box 24 (AT5100-0100)/XFB Inputs/Data <-> Data Pointer/HallSensorValues
//   Device 8 (EtherCAT) <-> TcCOM Objects/XTS ProcessingUnit 1/XL Part 3/XL Module 16
//     Box 25 (AT5100-0100)/DRV Commutation angle/Commutation angle <-> Data Pointer/CommutationAngle
//     Box 25 (AT5100-0100)/DRV Controlword/Controlword <-> Data Pointer/Control
//     Box 25 (AT5100-0100)/DRV Statusword/Statusword <-> Data Pointer/Status
//     Box 25 (AT5100-0100)/DRV Target torque/Target torque <-> Data Pointer/Torque
//     Box 25 (AT5100-0100)/XFB Inputs/Data <-> Data Pointer/HallSensorValues
//   Device 8 (EtherCAT) <-> TcCOM Objects/XTS ProcessingUnit 1/XL Part 3/XL Module 17
//     Box 26 (AT5100-0100)/DRV Commutation angle/Commutation angle <-> Data Pointer/CommutationAngle
//     Box 26 (AT5100-0100)/DRV Controlword/Controlword <-> Data Pointer/Control
//     Box 26 (AT5100-0100)/DRV Statusword/Statusword <-> Data Pointer/Status
//     Box 26 (AT5100-0100)/DRV Target torque/Target torque <-> Data Pointer/Torque
//     Box 26 (AT5100-0100)/XFB Inputs/Data <-> Data Pointer/HallSensorValues
//   Device 8 (EtherCAT) <-> TcCOM Objects/XTS ProcessingUnit 1/XL Part 3/XL Module 18
//     Box 27 (AT5100-0100)/DRV Commutation angle/Commutation angle <-> Data Pointer/CommutationAngle
//     Box 27 (AT5100-0100)/DRV Controlword/Controlword <-> Data Pointer/Control
//     Box 27 (AT5100-0100)/DRV Statusword/Statusword <-> Data Pointer/Status
//     Box 27 (AT5100-0100)/DRV Target torque/Target torque <-> Data Pointer/Torque
//     Box 27 (AT5100-0100)/XFB Inputs/Data <-> Data Pointer/HallSensorValues
//   Device 8 (EtherCAT) <-> TcCOM Objects/XTS ProcessingUnit 1/XL Part 3/XL Module 9
//     Box 18 (AT5100-0100)/DRV Commutation angle/Commutation angle <-> Data Pointer/CommutationAngle
//     Box 18 (AT5100-0100)/DRV Controlword/Controlword <-> Data Pointer/Control
//     Box 18 (AT5100-0100)/DRV Statusword/Statusword <-> Data Pointer/Status
//     Box 18 (AT5100-0100)/DRV Target torque/Target torque <-> Data Pointer/Torque
//     Box 18 (AT5100-0100)/XFB Inputs/Data <-> Data Pointer/HallSensorValues
//   PlanarTrackMovement_1/PlanarTrackMovement_1 Instance <-> Device 1 (EtherCAT)/Term 1 (EK1200)/Term 13 (EL2912)
//     PlcTask Inputs/MAIN.MoverStop <-> StandardInputs/TwinSafeGroup1.E-StopReq_139
//     PlcTask Outputs/MAIN.MoverStopDone <-> StandardOutputs/TwinSafeGroup1.STO_Release_140
//   PlanarTrackMovement_1/PlanarTrackMovement_1 Instance <-> Device 1 (EtherCAT)/Term 1 (EK1200)/Term 4 (EL2809)
//     PlcTask Outputs/MAIN.ResetSafetyLight <-> Channel 16/Output
//   PlanarTrackMovement_1/PlanarTrackMovement_1 Instance <-> Device 1 (EtherCAT)/Term 1 (EK1200)/Term 7 (EL4034)
//     PlcTask Outputs/GVL_General.stSwitchStatus.MagnetValue <-> AO Outputs Channel 1/Analog output
//   PlanarTrackMovement_1/PlanarTrackMovement_1 Instance <-> MC Project1/Axes/MC_Mover 1
//     PlcTask Inputs/GVL_Mc3.fbPlanarXtsMover[1]._McPlanarMover.MCTOPLC/ACT <-> McToPlc/ACT
//     PlcTask Inputs/GVL_Mc3.fbPlanarXtsMover[1]._McPlanarMover.MCTOPLC/COORDMODE <-> McToPlc/COORDMODE
//     PlcTask Inputs/GVL_Mc3.fbPlanarXtsMover[1]._McPlanarMover.MCTOPLC/SET <-> McToPlc/SET
//     PlcTask Inputs/GVL_Mc3.fbPlanarXtsMover[1]._McPlanarMover.MCTOPLC/SETONTRACK <-> McToPlc/SETONTRACK
//     PlcTask Inputs/GVL_Mc3.fbPlanarXtsMover[1]._McPlanarMover.MCTOPLC/STD <-> McToPlc/STD
//     PlcTask Outputs/GVL_Mc3.fbPlanarXtsMover[1]._McPlanarMover.PLCTOMC/STD <-> PlcToMc/STD
//   PlanarTrackMovement_1/PlanarTrackMovement_1 Instance <-> MC Project1/Axes/MC_Mover 2
//     PlcTask Inputs/GVL_Mc3.fbPlanarXtsMover[2]._McPlanarMover.MCTOPLC/ACT <-> McToPlc/ACT
//     PlcTask Inputs/GVL_Mc3.fbPlanarXtsMover[2]._McPlanarMover.MCTOPLC/COORDMODE <-> McToPlc/COORDMODE
//     PlcTask Inputs/GVL_Mc3.fbPlanarXtsMover[2]._McPlanarMover.MCTOPLC/SET <-> McToPlc/SET
//     PlcTask Inputs/GVL_Mc3.fbPlanarXtsMover[2]._McPlanarMover.MCTOPLC/SETONTRACK <-> McToPlc/SETONTRACK
//     PlcTask Inputs/GVL_Mc3.fbPlanarXtsMover[2]._McPlanarMover.MCTOPLC/STD <-> McToPlc/STD
//     PlcTask Outputs/GVL_Mc3.fbPlanarXtsMover[2]._McPlanarMover.PLCTOMC/STD <-> PlcToMc/STD
//   PlanarTrackMovement_1/PlanarTrackMovement_1 Instance <-> MC Project1/Axes/MC_Mover 3
//     PlcTask Inputs/GVL_Mc3.fbPlanarXtsMover[3]._McPlanarMover.MCTOPLC/ACT <-> McToPlc/ACT
//     PlcTask Inputs/GVL_Mc3.fbPlanarXtsMover[3]._McPlanarMover.MCTOPLC/COORDMODE <-> McToPlc/COORDMODE
//     PlcTask Inputs/GVL_Mc3.fbPlanarXtsMover[3]._McPlanarMover.MCTOPLC/SET <-> McToPlc/SET
//     PlcTask Inputs/GVL_Mc3.fbPlanarXtsMover[3]._McPlanarMover.MCTOPLC/SETONTRACK <-> McToPlc/SETONTRACK
//     PlcTask Inputs/GVL_Mc3.fbPlanarXtsMover[3]._McPlanarMover.MCTOPLC/STD <-> McToPlc/STD
//     PlcTask Outputs/GVL_Mc3.fbPlanarXtsMover[3]._McPlanarMover.PLCTOMC/STD <-> PlcToMc/STD
//   PlanarTrackMovement_1/PlanarTrackMovement_1 Instance <-> MC Project1/Axes/MC_Mover 4
//     PlcTask Inputs/GVL_Mc3.fbPlanarXtsMover[4]._McPlanarMover.MCTOPLC/ACT <-> McToPlc/ACT
//     PlcTask Inputs/GVL_Mc3.fbPlanarXtsMover[4]._McPlanarMover.MCTOPLC/COORDMODE <-> McToPlc/COORDMODE
//     PlcTask Inputs/GVL_Mc3.fbPlanarXtsMover[4]._McPlanarMover.MCTOPLC/SET <-> McToPlc/SET
//     PlcTask Inputs/GVL_Mc3.fbPlanarXtsMover[4]._McPlanarMover.MCTOPLC/SETONTRACK <-> McToPlc/SETONTRACK
//     PlcTask Inputs/GVL_Mc3.fbPlanarXtsMover[4]._McPlanarMover.MCTOPLC/STD <-> McToPlc/STD
//     PlcTask Outputs/GVL_Mc3.fbPlanarXtsMover[4]._McPlanarMover.PLCTOMC/STD <-> PlcToMc/STD
//   PlanarTrackMovement_1/PlanarTrackMovement_1 Instance <-> MC Project1/Groups/McTrack1
//     PlcTask Inputs/GVL_Mc3.MC_Tracks[1].MCTOPLC_STD <-> McToPlc/STD
//   PlanarTrackMovement_1/PlanarTrackMovement_1 Instance <-> MC Project1/Groups/McTrack2
//     PlcTask Inputs/GVL_Mc3.MC_Tracks[2].MCTOPLC_STD <-> McToPlc/STD
//   PlanarTrackMovement_1/PlanarTrackMovement_1 Instance <-> MC Project1/Groups/McTrack3
//     PlcTask Inputs/GVL_Mc3.MC_Tracks[3].MCTOPLC_STD <-> McToPlc/STD
//   SaftyPLC_1/SaftyPLC_1 Instance <-> Device 1 (EtherCAT)/Term 1 (EK1200)/Term 13 (EL2912)
//     PlcTask Inputs/GVL_Safety.Error_Com <-> StandardInputs/TwinSafeGroup1.Error_Com_142
//     PlcTask Inputs/GVL_Safety.Error_Other <-> StandardInputs/TwinSafeGroup1.Error_Other_143
//     PlcTask Inputs/GVL_Safety.Error_Out <-> StandardInputs/TwinSafeGroup1.Error_out_141
//     PlcTask Inputs/GVL_Safety.SaeftyOk <-> StandardInputs/TwinSafeGroup1.SafetyOk_72
//     PlcTask Inputs/GVL_Safety.SafetyInRun <-> StandardInputs/TwinSafeGroup1.SafetyInRun_73
//     PlcTask Outputs/GVL_Safety.Reset <-> StandardOutputs/TwinSafeGroup1.ErrorAcknowledgement_1
//     PlcTask Outputs/GVL_Safety.Run <-> StandardOutputs/TwinSafeGroup1.Run_2
//     PlcTask Outputs/GVL_Safety.Start <-> StandardOutputs/TwinSafeGroup1.STO_75
//   SaftyPLC_1/SaftyPLC_1 Instance <-> Device 1 (EtherCAT)/Term 1 (EK1200)/Term 2 (EL1809)
//     PlcTask Inputs/GVL_Safety.HwReset <-> Channel 16/Input
//     PlcTask Inputs/GVL_Safety.HwStart <-> Channel 14/Input
//     PlcTask Inputs/GVL_Safety.HwStop <-> Channel 15/Input
//   SaftyPLC_1/SaftyPLC_1 Instance <-> Device 4 (EtherCAT)/Box 50 (AT5100-0100)
//     PlcTask Inputs/GVL_io.D_Spannung[5] <-> DRV Info data 1/D-Spannung
//     PlcTask Inputs/GVL_io.Q_Spannung[5] <-> DRV Info data 1/Q-Spannung
//     PlcTask Outputs/GVL_Safety.Reset <-> Module 1 (SAFETY)/SAFETY Standard Outputdata/Standard In Var 1
//     PlcTask Outputs/GVL_Safety.Run <-> Module 1 (SAFETY)/SAFETY Standard Outputdata/Standard In Var 5
//   SaftyPLC_1/SaftyPLC_1 Instance <-> Device 4 (EtherCAT)/Box 51 (AT5100-0100)
//     PlcTask Inputs/GVL_io.D_Spannung[6] <-> DRV Info data 1/D-Spannung
//     PlcTask Inputs/GVL_io.Q_Spannung[6] <-> DRV Info data 1/Q-Spannung
//     PlcTask Outputs/GVL_Safety.Reset <-> Module 1 (SAFETY)/SAFETY Standard Outputdata/Standard In Var 1
//     PlcTask Outputs/GVL_Safety.Run <-> Module 1 (SAFETY)/SAFETY Standard Outputdata/Standard In Var 5
//   SaftyPLC_1/SaftyPLC_1 Instance <-> Device 4 (EtherCAT)/Box 52 (AT5100-0100)
//     PlcTask Outputs/GVL_Safety.Reset <-> Module 1 (SAFETY)/SAFETY Standard Outputdata/Standard In Var 1
//     PlcTask Outputs/GVL_Safety.Run <-> Module 1 (SAFETY)/SAFETY Standard Outputdata/Standard In Var 5
//   SaftyPLC_1/SaftyPLC_1 Instance <-> Device 4 (EtherCAT)/Box 53 (AT5100-0100)
//     PlcTask Outputs/GVL_Safety.Reset <-> Module 1 (SAFETY)/SAFETY Standard Outputdata/Standard In Var 1
//     PlcTask Outputs/GVL_Safety.Run <-> Module 1 (SAFETY)/SAFETY Standard Outputdata/Standard In Var 5
//   SaftyPLC_1/SaftyPLC_1 Instance <-> Device 4 (EtherCAT)/Box 54 (AT5100-0100)
//     PlcTask Outputs/GVL_Safety.Reset <-> Module 1 (SAFETY)/SAFETY Standard Outputdata/Standard In Var 1
//     PlcTask Outputs/GVL_Safety.Run <-> Module 1 (SAFETY)/SAFETY Standard Outputdata/Standard In Var 5
//   SaftyPLC_1/SaftyPLC_1 Instance <-> Device 4 (EtherCAT)/Box 55 (AT5100-0100)
//     PlcTask Outputs/GVL_Safety.Reset <-> Module 1 (SAFETY)/SAFETY Standard Outputdata/Standard In Var 1
//     PlcTask Outputs/GVL_Safety.Run <-> Module 1 (SAFETY)/SAFETY Standard Outputdata/Standard In Var 5
//   SaftyPLC_1/SaftyPLC_1 Instance <-> Device 4 (EtherCAT)/Box 56 (AT5100-0100)
//     PlcTask Outputs/GVL_Safety.Reset <-> Module 1 (SAFETY)/SAFETY Standard Outputdata/Standard In Var 1
//     PlcTask Outputs/GVL_Safety.Run <-> Module 1 (SAFETY)/SAFETY Standard Outputdata/Standard In Var 5
//   SaftyPLC_1/SaftyPLC_1 Instance <-> Device 4 (EtherCAT)/Box 57 (AT5100-0100)
//     PlcTask Outputs/GVL_Safety.Reset <-> Module 1 (SAFETY)/SAFETY Standard Outputdata/Standard In Var 1
//     PlcTask Outputs/GVL_Safety.Run <-> Module 1 (SAFETY)/SAFETY Standard Outputdata/Standard In Var 5
//   SaftyPLC_1/SaftyPLC_1 Instance <-> Device 4 (EtherCAT)/Box 58 (AT5100-0100)
//     PlcTask Outputs/GVL_Safety.Reset <-> Module 1 (SAFETY)/SAFETY Standard Outputdata/Standard In Var 1
//     PlcTask Outputs/GVL_Safety.Run <-> Module 1 (SAFETY)/SAFETY Standard Outputdata/Standard In Var 5
//   SaftyPLC_1/SaftyPLC_1 Instance <-> Device 4 (EtherCAT)/Box 59 (AT5100-0100)
//     PlcTask Outputs/GVL_Safety.Reset <-> Module 1 (SAFETY)/SAFETY Standard Outputdata/Standard In Var 1
//     PlcTask Outputs/GVL_Safety.Run <-> Module 1 (SAFETY)/SAFETY Standard Outputdata/Standard In Var 5
//   SaftyPLC_1/SaftyPLC_1 Instance <-> Device 4 (EtherCAT)/Box 60 (AT5100-0100)
//     PlcTask Outputs/GVL_Safety.Reset <-> Module 1 (SAFETY)/SAFETY Standard Outputdata/Standard In Var 1
//     PlcTask Outputs/GVL_Safety.Run <-> Module 1 (SAFETY)/SAFETY Standard Outputdata/Standard In Var 5
//   SaftyPLC_1/SaftyPLC_1 Instance <-> Device 4 (EtherCAT)/Box 61 (AT5100-0100)
//     PlcTask Outputs/GVL_Safety.Reset <-> Module 1 (SAFETY)/SAFETY Standard Outputdata/Standard In Var 1
//     PlcTask Outputs/GVL_Safety.Run <-> Module 1 (SAFETY)/SAFETY Standard Outputdata/Standard In Var 5
//   SaftyPLC_1/SaftyPLC_1 Instance <-> Device 4 (EtherCAT)/Box 62 (AT5100-0100)
//     PlcTask Outputs/GVL_Safety.Reset <-> Module 1 (SAFETY)/SAFETY Standard Outputdata/Standard In Var 1
//     PlcTask Outputs/GVL_Safety.Run <-> Module 1 (SAFETY)/SAFETY Standard Outputdata/Standard In Var 5
//   SaftyPLC_1/SaftyPLC_1 Instance <-> Device 4 (EtherCAT)/Box 63 (AT5100-0100)
//     PlcTask Outputs/GVL_Safety.Reset <-> Module 1 (SAFETY)/SAFETY Standard Outputdata/Standard In Var 1
//     PlcTask Outputs/GVL_Safety.Run <-> Module 1 (SAFETY)/SAFETY Standard Outputdata/Standard In Var 5
//   SaftyPLC_1/SaftyPLC_1 Instance <-> Device 4 (EtherCAT)/Box 64 (AT5100-0100)
//     PlcTask Outputs/GVL_Safety.Reset <-> Module 1 (SAFETY)/SAFETY Standard Outputdata/Standard In Var 1
//     PlcTask Outputs/GVL_Safety.Run <-> Module 1 (SAFETY)/SAFETY Standard Outputdata/Standard In Var 5
//   SaftyPLC_1/SaftyPLC_1 Instance <-> Device 4 (EtherCAT)/Box 65 (AT5100-0100)
//     PlcTask Outputs/GVL_Safety.Reset <-> Module 1 (SAFETY)/SAFETY Standard Outputdata/Standard In Var 1
//     PlcTask Outputs/GVL_Safety.Run <-> Module 1 (SAFETY)/SAFETY Standard Outputdata/Standard In Var 5
//   SaftyPLC_1/SaftyPLC_1 Instance <-> Device 4 (EtherCAT)/Box 66 (AT5100-0100)
//     PlcTask Outputs/GVL_Safety.Reset <-> Module 1 (SAFETY)/SAFETY Standard Outputdata/Standard In Var 1
//     PlcTask Outputs/GVL_Safety.Run <-> Module 1 (SAFETY)/SAFETY Standard Outputdata/Standard In Var 5
//   SaftyPLC_1/SaftyPLC_1 Instance <-> Device 4 (EtherCAT)/Box 67 (AT5100-0100)
//     PlcTask Outputs/GVL_Safety.Reset <-> Module 1 (SAFETY)/SAFETY Standard Outputdata/Standard In Var 1
//     PlcTask Outputs/GVL_Safety.Run <-> Module 1 (SAFETY)/SAFETY Standard Outputdata/Standard In Var 5
//   SaftyPLC_1/SaftyPLC_1 Instance <-> Device 4 (EtherCAT)/Box 68 (AT5100-0100)
//     PlcTask Outputs/GVL_Safety.Reset <-> Module 1 (SAFETY)/SAFETY Standard Outputdata/Standard In Var 1
//     PlcTask Outputs/GVL_Safety.Run <-> Module 1 (SAFETY)/SAFETY Standard Outputdata/Standard In Var 5
//   SaftyPLC_1/SaftyPLC_1 Instance <-> Device 4 (EtherCAT)/Box 69 (AT5100-0100)
//     PlcTask Outputs/GVL_Safety.Reset <-> Module 1 (SAFETY)/SAFETY Standard Outputdata/Standard In Var 1
//     PlcTask Outputs/GVL_Safety.Run <-> Module 1 (SAFETY)/SAFETY Standard Outputdata/Standard In Var 5
//   SaftyPLC_1/SaftyPLC_1 Instance <-> Device 4 (EtherCAT)/Box 70 (AT5100-0100)
//     PlcTask Outputs/GVL_Safety.Reset <-> Module 1 (SAFETY)/SAFETY Standard Outputdata/Standard In Var 1
//     PlcTask Outputs/GVL_Safety.Run <-> Module 1 (SAFETY)/SAFETY Standard Outputdata/Standard In Var 5
//   SaftyPLC_1/SaftyPLC_1 Instance <-> Device 4 (EtherCAT)/Box 71 (AT5100-0100)
//     PlcTask Outputs/GVL_Safety.Reset <-> Module 1 (SAFETY)/SAFETY Standard Outputdata/Standard In Var 1
//     PlcTask Outputs/GVL_Safety.Run <-> Module 1 (SAFETY)/SAFETY Standard Outputdata/Standard In Var 5
//   SaftyPLC_1/SaftyPLC_1 Instance <-> Device 4 (EtherCAT)/Box 72 (AT5100-0100)
//     PlcTask Outputs/GVL_Safety.Reset <-> Module 1 (SAFETY)/SAFETY Standard Outputdata/Standard In Var 1
//     PlcTask Outputs/GVL_Safety.Run <-> Module 1 (SAFETY)/SAFETY Standard Outputdata/Standard In Var 5
//   SaftyPLC_1/SaftyPLC_1 Instance <-> Device 4 (EtherCAT)/Box 73 (AT5100-0100)
//     PlcTask Outputs/GVL_Safety.Reset <-> Module 1 (SAFETY)/SAFETY Standard Outputdata/Standard In Var 1
//     PlcTask Outputs/GVL_Safety.Run <-> Module 1 (SAFETY)/SAFETY Standard Outputdata/Standard In Var 5
//   SaftyPLC_1/SaftyPLC_1 Instance <-> Device 4 (EtherCAT)/Box 74 (AT5100-0100)
//     PlcTask Outputs/GVL_Safety.Reset <-> Module 1 (SAFETY)/SAFETY Standard Outputdata/Standard In Var 1
//     PlcTask Outputs/GVL_Safety.Run <-> Module 1 (SAFETY)/SAFETY Standard Outputdata/Standard In Var 5
//   SaftyPLC_1/SaftyPLC_1 Instance <-> Device 4 (EtherCAT)/Box 75 (AT5100-0100)
//     PlcTask Outputs/GVL_Safety.Reset <-> Module 1 (SAFETY)/SAFETY Standard Outputdata/Standard In Var 1
//     PlcTask Outputs/GVL_Safety.Run <-> Module 1 (SAFETY)/SAFETY Standard Outputdata/Standard In Var 5
//   SaftyPLC_1/SaftyPLC_1 Instance <-> Device 4 (EtherCAT)/Box 76 (AT5100-0100)
//     PlcTask Outputs/GVL_Safety.Reset <-> Module 1 (SAFETY)/SAFETY Standard Outputdata/Standard In Var 1
//     PlcTask Outputs/GVL_Safety.Run <-> Module 1 (SAFETY)/SAFETY Standard Outputdata/Standard In Var 5
//   SaftyPLC_1/SaftyPLC_1 Instance <-> Device 4 (EtherCAT)/Box 77 (AT5100-0100)
//     PlcTask Outputs/GVL_Safety.Reset <-> Module 1 (SAFETY)/SAFETY Standard Outputdata/Standard In Var 1
//     PlcTask Outputs/GVL_Safety.Run <-> Module 1 (SAFETY)/SAFETY Standard Outputdata/Standard In Var 5
//   SaftyPLC_1/SaftyPLC_1 Instance <-> Device 4 (EtherCAT)/Box 78 (AT5100-0100)
//     PlcTask Outputs/GVL_Safety.Reset <-> Module 1 (SAFETY)/SAFETY Standard Outputdata/Standard In Var 1
//     PlcTask Outputs/GVL_Safety.Run <-> Module 1 (SAFETY)/SAFETY Standard Outputdata/Standard In Var 5
//   SaftyPLC_1/SaftyPLC_1 Instance <-> Device 4 (EtherCAT)/Box 79 (AT5100-0100)
//     PlcTask Outputs/GVL_Safety.Reset <-> Module 1 (SAFETY)/SAFETY Standard Outputdata/Standard In Var 1
//     PlcTask Outputs/GVL_Safety.Run <-> Module 1 (SAFETY)/SAFETY Standard Outputdata/Standard In Var 5
//   SaftyPLC_1/SaftyPLC_1 Instance <-> Device 4 (EtherCAT)/Box 80 (AT5100-0100)
//     PlcTask Inputs/GVL_io.D_Spannung[7] <-> DRV Info data 1/D-Spannung
//     PlcTask Inputs/GVL_io.Q_Spannung[7] <-> DRV Info data 1/Q-Spannung
//     PlcTask Outputs/GVL_Safety.Reset <-> Module 1 (SAFETY)/SAFETY Standard Outputdata/Standard In Var 1
//     PlcTask Outputs/GVL_Safety.Run <-> Module 1 (SAFETY)/SAFETY Standard Outputdata/Standard In Var 5
//   SaftyPLC_1/SaftyPLC_1 Instance <-> Device 4 (EtherCAT)/Box 81 (AT5100-0100)
//     PlcTask Inputs/GVL_io.D_Spannung[8] <-> DRV Info data 1/D-Spannung
//     PlcTask Inputs/GVL_io.Q_Spannung[8] <-> DRV Info data 1/Q-Spannung
//     PlcTask Outputs/GVL_Safety.Reset <-> Module 1 (SAFETY)/SAFETY Standard Outputdata/Standard In Var 1
//     PlcTask Outputs/GVL_Safety.Run <-> Module 1 (SAFETY)/SAFETY Standard Outputdata/Standard In Var 5
//   SaftyPLC_1/SaftyPLC_1 Instance <-> Device 8 (EtherCAT)/Box 18 (AT5100-0100)
//     PlcTask Inputs/GVL_io.D_Spannung[1] <-> DRV Info data 1/D-Spannung
//     PlcTask Inputs/GVL_io.Q_Spannung[1] <-> DRV Info data 1/Q-Spannung
//     PlcTask Outputs/GVL_Safety.Reset <-> Module 1 (SAFETY)/SAFETY Standard Outputdata/Standard In Var 1
//     PlcTask Outputs/GVL_Safety.Run <-> Module 1 (SAFETY)/SAFETY Standard Outputdata/Standard In Var 5
//   SaftyPLC_1/SaftyPLC_1 Instance <-> Device 8 (EtherCAT)/Box 19 (AT5100-0100)
//     PlcTask Inputs/GVL_io.D_Spannung[2] <-> DRV Info data 1/D-Spannung
//     PlcTask Inputs/GVL_io.Q_Spannung[2] <-> DRV Info data 1/Q-Spannung
//     PlcTask Outputs/GVL_Safety.Reset <-> Module 1 (SAFETY)/SAFETY Standard Outputdata/Standard In Var 1
//     PlcTask Outputs/GVL_Safety.Run <-> Module 1 (SAFETY)/SAFETY Standard Outputdata/Standard In Var 5
//   SaftyPLC_1/SaftyPLC_1 Instance <-> Device 8 (EtherCAT)/Box 20 (AT5100-0100)
//     PlcTask Outputs/GVL_Safety.Reset <-> Module 1 (SAFETY)/SAFETY Standard Outputdata/Standard In Var 1
//     PlcTask Outputs/GVL_Safety.Run <-> Module 1 (SAFETY)/SAFETY Standard Outputdata/Standard In Var 5
//   SaftyPLC_1/SaftyPLC_1 Instance <-> Device 8 (EtherCAT)/Box 21 (AT5100-0100)
//     PlcTask Outputs/GVL_Safety.Reset <-> Module 1 (SAFETY)/SAFETY Standard Outputdata/Standard In Var 1
//     PlcTask Outputs/GVL_Safety.Run <-> Module 1 (SAFETY)/SAFETY Standard Outputdata/Standard In Var 5
//   SaftyPLC_1/SaftyPLC_1 Instance <-> Device 8 (EtherCAT)/Box 22 (AT5100-0100)
//     PlcTask Outputs/GVL_Safety.Reset <-> Module 1 (SAFETY)/SAFETY Standard Outputdata/Standard In Var 1
//     PlcTask Outputs/GVL_Safety.Run <-> Module 1 (SAFETY)/SAFETY Standard Outputdata/Standard In Var 5
//   SaftyPLC_1/SaftyPLC_1 Instance <-> Device 8 (EtherCAT)/Box 23 (AT5100-0100)
//     PlcTask Outputs/GVL_Safety.Reset <-> Module 1 (SAFETY)/SAFETY Standard Outputdata/Standard In Var 1
//     PlcTask Outputs/GVL_Safety.Run <-> Module 1 (SAFETY)/SAFETY Standard Outputdata/Standard In Var 5
//   SaftyPLC_1/SaftyPLC_1 Instance <-> Device 8 (EtherCAT)/Box 24 (AT5100-0100)
//     PlcTask Outputs/GVL_Safety.Reset <-> Module 1 (SAFETY)/SAFETY Standard Outputdata/Standard In Var 1
//     PlcTask Outputs/GVL_Safety.Run <-> Module 1 (SAFETY)/SAFETY Standard Outputdata/Standard In Var 5
//   SaftyPLC_1/SaftyPLC_1 Instance <-> Device 8 (EtherCAT)/Box 25 (AT5100-0100)
//     PlcTask Outputs/GVL_Safety.Reset <-> Module 1 (SAFETY)/SAFETY Standard Outputdata/Standard In Var 1
//     PlcTask Outputs/GVL_Safety.Run <-> Module 1 (SAFETY)/SAFETY Standard Outputdata/Standard In Var 5
//   SaftyPLC_1/SaftyPLC_1 Instance <-> Device 8 (EtherCAT)/Box 26 (AT5100-0100)
//     PlcTask Outputs/GVL_Safety.Reset <-> Module 1 (SAFETY)/SAFETY Standard Outputdata/Standard In Var 1
//     PlcTask Outputs/GVL_Safety.Run <-> Module 1 (SAFETY)/SAFETY Standard Outputdata/Standard In Var 5
//   SaftyPLC_1/SaftyPLC_1 Instance <-> Device 8 (EtherCAT)/Box 27 (AT5100-0100)
//     PlcTask Outputs/GVL_Safety.Reset <-> Module 1 (SAFETY)/SAFETY Standard Outputdata/Standard In Var 1
//     PlcTask Outputs/GVL_Safety.Run <-> Module 1 (SAFETY)/SAFETY Standard Outputdata/Standard In Var 5
//   SaftyPLC_1/SaftyPLC_1 Instance <-> Device 8 (EtherCAT)/Box 28 (AT5100-0100)
//     PlcTask Outputs/GVL_Safety.Reset <-> Module 1 (SAFETY)/SAFETY Standard Outputdata/Standard In Var 1
//     PlcTask Outputs/GVL_Safety.Run <-> Module 1 (SAFETY)/SAFETY Standard Outputdata/Standard In Var 5
//   SaftyPLC_1/SaftyPLC_1 Instance <-> Device 8 (EtherCAT)/Box 29 (AT5100-0100)
//     PlcTask Outputs/GVL_Safety.Reset <-> Module 1 (SAFETY)/SAFETY Standard Outputdata/Standard In Var 1
//     PlcTask Outputs/GVL_Safety.Run <-> Module 1 (SAFETY)/SAFETY Standard Outputdata/Standard In Var 5
//   SaftyPLC_1/SaftyPLC_1 Instance <-> Device 8 (EtherCAT)/Box 30 (AT5100-0100)
//     PlcTask Outputs/GVL_Safety.Reset <-> Module 1 (SAFETY)/SAFETY Standard Outputdata/Standard In Var 1
//     PlcTask Outputs/GVL_Safety.Run <-> Module 1 (SAFETY)/SAFETY Standard Outputdata/Standard In Var 5
//   SaftyPLC_1/SaftyPLC_1 Instance <-> Device 8 (EtherCAT)/Box 31 (AT5100-0100)
//     PlcTask Outputs/GVL_Safety.Reset <-> Module 1 (SAFETY)/SAFETY Standard Outputdata/Standard In Var 1
//     PlcTask Outputs/GVL_Safety.Run <-> Module 1 (SAFETY)/SAFETY Standard Outputdata/Standard In Var 5
//   SaftyPLC_1/SaftyPLC_1 Instance <-> Device 8 (EtherCAT)/Box 32 (AT5100-0100)
//     PlcTask Outputs/GVL_Safety.Reset <-> Module 1 (SAFETY)/SAFETY Standard Outputdata/Standard In Var 1
//     PlcTask Outputs/GVL_Safety.Run <-> Module 1 (SAFETY)/SAFETY Standard Outputdata/Standard In Var 5
//   SaftyPLC_1/SaftyPLC_1 Instance <-> Device 8 (EtherCAT)/Box 33 (AT5100-0100)
//     PlcTask Outputs/GVL_Safety.Reset <-> Module 1 (SAFETY)/SAFETY Standard Outputdata/Standard In Var 1
//     PlcTask Outputs/GVL_Safety.Run <-> Module 1 (SAFETY)/SAFETY Standard Outputdata/Standard In Var 5
//   SaftyPLC_1/SaftyPLC_1 Instance <-> Device 8 (EtherCAT)/Box 34 (AT5100-0100)
//     PlcTask Outputs/GVL_Safety.Reset <-> Module 1 (SAFETY)/SAFETY Standard Outputdata/Standard In Var 1
//     PlcTask Outputs/GVL_Safety.Run <-> Module 1 (SAFETY)/SAFETY Standard Outputdata/Standard In Var 5
//   SaftyPLC_1/SaftyPLC_1 Instance <-> Device 8 (EtherCAT)/Box 35 (AT5100-0100)
//     PlcTask Outputs/GVL_Safety.Reset <-> Module 1 (SAFETY)/SAFETY Standard Outputdata/Standard In Var 1
//     PlcTask Outputs/GVL_Safety.Run <-> Module 1 (SAFETY)/SAFETY Standard Outputdata/Standard In Var 5
//   SaftyPLC_1/SaftyPLC_1 Instance <-> Device 8 (EtherCAT)/Box 36 (AT5100-0100)
//     PlcTask Outputs/GVL_Safety.Reset <-> Module 1 (SAFETY)/SAFETY Standard Outputdata/Standard In Var 1
//     PlcTask Outputs/GVL_Safety.Run <-> Module 1 (SAFETY)/SAFETY Standard Outputdata/Standard In Var 5
//   SaftyPLC_1/SaftyPLC_1 Instance <-> Device 8 (EtherCAT)/Box 37 (AT5100-0100)
//     PlcTask Outputs/GVL_Safety.Reset <-> Module 1 (SAFETY)/SAFETY Standard Outputdata/Standard In Var 1
//     PlcTask Outputs/GVL_Safety.Run <-> Module 1 (SAFETY)/SAFETY Standard Outputdata/Standard In Var 5
//   SaftyPLC_1/SaftyPLC_1 Instance <-> Device 8 (EtherCAT)/Box 38 (AT5100-0100)
//     PlcTask Outputs/GVL_Safety.Reset <-> Module 1 (SAFETY)/SAFETY Standard Outputdata/Standard In Var 1
//     PlcTask Outputs/GVL_Safety.Run <-> Module 1 (SAFETY)/SAFETY Standard Outputdata/Standard In Var 5
//   SaftyPLC_1/SaftyPLC_1 Instance <-> Device 8 (EtherCAT)/Box 39 (AT5100-0100)
//     PlcTask Outputs/GVL_Safety.Reset <-> Module 1 (SAFETY)/SAFETY Standard Outputdata/Standard In Var 1
//     PlcTask Outputs/GVL_Safety.Run <-> Module 1 (SAFETY)/SAFETY Standard Outputdata/Standard In Var 5
//   SaftyPLC_1/SaftyPLC_1 Instance <-> Device 8 (EtherCAT)/Box 40 (AT5100-0100)
//     PlcTask Outputs/GVL_Safety.Reset <-> Module 1 (SAFETY)/SAFETY Standard Outputdata/Standard In Var 1
//     PlcTask Outputs/GVL_Safety.Run <-> Module 1 (SAFETY)/SAFETY Standard Outputdata/Standard In Var 5
//   SaftyPLC_1/SaftyPLC_1 Instance <-> Device 8 (EtherCAT)/Box 41 (AT5100-0100)
//     PlcTask Outputs/GVL_Safety.Reset <-> Module 1 (SAFETY)/SAFETY Standard Outputdata/Standard In Var 1
//     PlcTask Outputs/GVL_Safety.Run <-> Module 1 (SAFETY)/SAFETY Standard Outputdata/Standard In Var 5
//   SaftyPLC_1/SaftyPLC_1 Instance <-> Device 8 (EtherCAT)/Box 42 (AT5100-0100)
//     PlcTask Outputs/GVL_Safety.Reset <-> Module 1 (SAFETY)/SAFETY Standard Outputdata/Standard In Var 1
//     PlcTask Outputs/GVL_Safety.Run <-> Module 1 (SAFETY)/SAFETY Standard Outputdata/Standard In Var 5
//   SaftyPLC_1/SaftyPLC_1 Instance <-> Device 8 (EtherCAT)/Box 43 (AT5100-0100)
//     PlcTask Outputs/GVL_Safety.Reset <-> Module 1 (SAFETY)/SAFETY Standard Outputdata/Standard In Var 1
//     PlcTask Outputs/GVL_Safety.Run <-> Module 1 (SAFETY)/SAFETY Standard Outputdata/Standard In Var 5
//   SaftyPLC_1/SaftyPLC_1 Instance <-> Device 8 (EtherCAT)/Box 44 (AT5100-0100)
//     PlcTask Outputs/GVL_Safety.Reset <-> Module 1 (SAFETY)/SAFETY Standard Outputdata/Standard In Var 1
//     PlcTask Outputs/GVL_Safety.Run <-> Module 1 (SAFETY)/SAFETY Standard Outputdata/Standard In Var 5
//   SaftyPLC_1/SaftyPLC_1 Instance <-> Device 8 (EtherCAT)/Box 45 (AT5100-0100)
//     PlcTask Outputs/GVL_Safety.Reset <-> Module 1 (SAFETY)/SAFETY Standard Outputdata/Standard In Var 1
//     PlcTask Outputs/GVL_Safety.Run <-> Module 1 (SAFETY)/SAFETY Standard Outputdata/Standard In Var 5
//   SaftyPLC_1/SaftyPLC_1 Instance <-> Device 8 (EtherCAT)/Box 46 (AT5100-0100)
//     PlcTask Outputs/GVL_Safety.Reset <-> Module 1 (SAFETY)/SAFETY Standard Outputdata/Standard In Var 1
//     PlcTask Outputs/GVL_Safety.Run <-> Module 1 (SAFETY)/SAFETY Standard Outputdata/Standard In Var 5
//   SaftyPLC_1/SaftyPLC_1 Instance <-> Device 8 (EtherCAT)/Box 47 (AT5100-0100)
//     PlcTask Outputs/GVL_Safety.Reset <-> Module 1 (SAFETY)/SAFETY Standard Outputdata/Standard In Var 1
//     PlcTask Outputs/GVL_Safety.Run <-> Module 1 (SAFETY)/SAFETY Standard Outputdata/Standard In Var 5
//   SaftyPLC_1/SaftyPLC_1 Instance <-> Device 8 (EtherCAT)/Box 48 (AT5100-0100)
//     PlcTask Inputs/GVL_io.D_Spannung[3] <-> DRV Info data 1/D-Spannung
//     PlcTask Inputs/GVL_io.Q_Spannung[3] <-> DRV Info data 1/Q-Spannung
//     PlcTask Outputs/GVL_Safety.Reset <-> Module 1 (SAFETY)/SAFETY Standard Outputdata/Standard In Var 1
//     PlcTask Outputs/GVL_Safety.Run <-> Module 1 (SAFETY)/SAFETY Standard Outputdata/Standard In Var 5
//   SaftyPLC_1/SaftyPLC_1 Instance <-> Device 8 (EtherCAT)/Box 49 (AT5100-0100)
//     PlcTask Inputs/GVL_io.D_Spannung[4] <-> DRV Info data 1/D-Spannung
//     PlcTask Inputs/GVL_io.Q_Spannung[4] <-> DRV Info data 1/Q-Spannung
//     PlcTask Outputs/GVL_Safety.Reset <-> Module 1 (SAFETY)/SAFETY Standard Outputdata/Standard In Var 1
//     PlcTask Outputs/GVL_Safety.Run <-> Module 1 (SAFETY)/SAFETY Standard Outputdata/Standard In Var 5

CONFIGURATION PlanarTrackMovement_1
    RESOURCE PLC ON TwinCAT3
        TASK PlcTask(INTERVAL := T#1ms, PRIORITY := 20);
        PROGRAM MAIN WITH PlcTask : MAIN;
    END_RESOURCE
END_CONFIGURATION

// ---- DUTs/E_MergeType.TcDUT
{attribute 'qualified_only'}
{attribute 'strict'}
TYPE E_MergeType :
(
	NoMerge := 0,
	FlyingMergeMoveOnTrack,
	FlyingMergeMoveSyncd,
	MergeFromStaticSyncd
);
END_TYPE

// ---- DUTs/E_TrackNum.TcDUT
{attribute 'qualified_only'}
//{attribute 'strict'}
TYPE E_TrackNum :
(
	Big		:=1,
	Small	:=2,
	Main	:=3
);	
END_TYPE

// ---- DUTs/MoverSort.TcDUT
TYPE MoverSort :
STRUCT
	MoverNumber 	: UDINT;
	TrackID  		: PlanarTrackOTCID;
	MoverPos 		: LREAL;
	MoverTrackNr 	: UDINT;
END_STRUCT
END_TYPE

// ---- DUTs/ST_Debounce.TcDUT
TYPE ST_Debounce :
STRUCT
	RawSignal : BOOL;
	DebSignal : BOOL;
END_STRUCT
END_TYPE

// ---- DUTs/ST_MoverOptions.TcDUT
TYPE ST_MoverOptions :
STRUCT
	BaseMoveOptions						: REFERENCE TO Tc3_Mc3PlanarMotion.ST_MoveOnTrackOptions;
	GearInMasterMoverOptions	: REFERENCE TO Tc3_Mc3PlanarMotion.ST_GearInPosOnTrackWithMasterMoverOptions;
	TempGap 									: LREAL := stMoverConfig.TightMoverGap; //for ramping up/down gap over a sector
	OptionUpdateInterval			:	LREAL := 5.0; //mm
	GapInTransition						: BOOL;
	MasterSyncPosition				: LREAL;
	MasterMoverID							: UDINT;
END_STRUCT
END_TYPE

// ---- DUTs/ST_PlanarTrackConfig.TcDUT
TYPE ST_PlanarTrackConfig :
STRUCT
	TrackIndex	: E_TrackNum;
	MCTrack		: CDT_MCTOPLC_PLANAR_TRACK;
END_STRUCT
END_TYPE

